LIN {X 5.728,Y -46.480,Z -106.471,A -90.000,B 90.000,C 0.000} C_DIS
LIN {X 5.220,Y -46.443,Z -106.628,A -90.000,B 90.000,C 0.000} C_DIS
LIN {X 4.791,Y -46.421,Z -106.762,A -90.000,B 90.000,C 0.000} C_DIS
LIN {X 4.548,Y -46.408,Z -106.845,A -90.000,B 90.000,C 0.000} C_DIS
LIN {X 4.247,Y -46.392,Z -106.952,A -90.000,B 90.000,C 0.000} C_DIS
LIN {X 3.683,Y -46.360,Z -107.175,A -90.000,B 90.000,C 0.000} C_DIS
LIN {X 3.330,Y -46.340,Z -107.324,A -90.000,B 90.000,C 0.000} C_DIS
LIN {X 2.924,Y -46.316,Z -107.512,A -90.000,B 90.000,C 0.000} C_DIS
LIN {X 2.654,Y -46.295,Z -107.645,A -90.000,B 90.000,C 0.000} C_DIS
LIN {X 1.447,Y -46.195,Z -108.262,A -90.000,B 90.000,C 0.000} C_DIS
LIN {X -0.684,Y -46.006,Z -109.354,A -90.000,B 90.000,C 0.000} C_DIS
LIN {X -0.987,Y -45.980,Z -109.516,A -90.000,B 90.000,C 0.000} C_DIS
LIN {X -1.310,Y -45.954,Z -109.697,A -90.000,B 90.000,C 0.000} C_DIS
LIN {X -1.716,Y -45.921,Z -109.939,A -90.000,B 90.000,C 0.000} C_DIS
LIN {X -2.229,Y -45.880,Z -110.266,A -90.000,B 90.000,C 0.000} C_DIS
LIN {X -2.497,Y -45.855,Z -110.452,A -90.000,B 90.000,C 0.000} C_DIS
LIN {X -4.271,Y -45.671,Z -111.693,A -90.000,B 90.000,C 0.000} C_DIS
LIN {X -4.661,Y -45.624,Z -111.967,A -90.000,B 90.000,C 0.000} C_DIS
LIN {X -5.221,Y -45.555,Z -112.383,A -90.000,B 90.000,C 0.000} C_DIS
LIN {X -5.480,Y -45.523,Z -112.584,A -90.000,B 90.000,C 0.000} C_DIS
LIN {X -5.669,Y -45.500,Z -112.740,A -90.000,B 90.000,C 0.000} C_DIS
LIN {X -5.871,Y -45.470,Z -112.907,A -90.000,B 90.000,C 0.000} C_DIS
LIN {X -6.143,Y -45.427,Z -113.144,A -90.000,B 90.000,C 0.000} C_DIS
LIN {X -6.336,Y -45.396,Z -113.323,A -90.000,B 90.000,C 0.000} C_DIS
LIN {X -7.007,Y -45.308,Z -113.952,A -90.000,B 90.000,C 0.000} C_DIS
LIN {X -7.165,Y -45.288,Z -114.092,A -90.000,B 90.000,C 0.000} C_DIS
LIN {X -7.242,Y -45.278,Z -114.154,A -90.000,B 90.000,C 0.000} C_DIS
LIN {X -7.389,Y -45.260,Z -114.260,A -90.000,B 90.000,C 0.000} C_DIS
LIN {X -7.460,Y -45.251,Z -114.305,A -90.000,B 90.000,C 0.000} C_DIS
LIN {X -7.595,Y -45.234,Z -114.380,A -90.000,B 90.000,C 0.000} C_DIS
LIN {X -7.660,Y -45.226,Z -114.410,A -90.000,B 90.000,C 0.000} C_DIS
LIN {X -7.783,Y -45.212,Z -114.455,A -90.000,B 90.000,C 0.000} C_DIS
LIN {X -7.869,Y -45.202,Z -114.476,A -90.000,B 90.000,C 0.000} C_DIS
LIN {X -7.951,Y -45.193,Z -114.487,A -90.000,B 90.000,C 0.000} C_DIS
LIN {X -8.029,Y -45.184,Z -114.489,A -90.000,B 90.000,C 0.000} C_DIS
LIN {X -8.077,Y -45.179,Z -114.485,A -90.000,B 90.000,C 0.000} C_DIS
LIN {X -8.124,Y -45.174,Z -114.476,A -90.000,B 90.000,C 0.000} C_DIS
LIN {X -8.189,Y -45.167,Z -114.456,A -90.000,B 90.000,C 0.000} C_DIS
LIN {X -8.249,Y -45.161,Z -114.428,A -90.000,B 90.000,C 0.000} C_DIS
LIN {X -8.305,Y -45.156,Z -114.391,A -90.000,B 90.000,C 0.000} C_DIS
LIN {X -8.338,Y -45.153,Z -114.363,A -90.000,B 90.000,C 0.000} C_DIS
LIN {X -8.370,Y -45.150,Z -114.331,A -90.000,B 90.000,C 0.000} C_DIS
LIN {X -8.425,Y -45.146,Z -114.257,A -90.000,B 90.000,C 0.000} C_DIS
LIN {X -8.450,Y -45.144,Z -114.216,A -90.000,B 90.000,C 0.000} C_DIS
LIN {X -8.490,Y -45.142,Z -114.125,A -90.000,B 90.000,C 0.000} C_DIS
LIN {X -8.507,Y -45.141,Z -114.075,A -90.000,B 90.000,C 0.000} C_DIS
LIN {X -8.533,Y -45.140,Z -113.968,A -90.000,B 90.000,C 0.000} C_DIS
LIN {X -8.548,Y -45.141,Z -113.852,A -90.000,B 90.000,C 0.000} C_DIS
LIN {X -8.552,Y -45.142,Z -113.791,A -90.000,B 90.000,C 0.000} C_DIS
LIN {X -8.552,Y -45.145,Z -113.662,A -90.000,B 90.000,C 0.000} C_DIS
LIN {X -8.547,Y -45.147,Z -113.595,A -90.000,B 90.000,C 0.000} C_DIS
LIN {X -8.531,Y -45.151,Z -113.457,A -90.000,B 90.000,C 0.000} C_DIS
LIN {X -8.518,Y -45.154,Z -113.385,A -90.000,B 90.000,C 0.000} C_DIS
LIN {X -8.485,Y -45.161,Z -113.238,A -90.000,B 90.000,C 0.000} C_DIS
LIN {X -8.464,Y -45.165,Z -113.163,A -90.000,B 90.000,C 0.000} C_DIS
LIN {X -8.414,Y -45.173,Z -113.010,A -90.000,B 90.000,C 0.000} C_DIS
LIN {X -8.352,Y -45.183,Z -112.854,A -90.000,B 90.000,C 0.000} C_DIS
LIN {X -8.316,Y -45.188,Z -112.775,A -90.000,B 90.000,C 0.000} C_DIS
LIN {X -8.236,Y -45.200,Z -112.616,A -90.000,B 90.000,C 0.000} C_DIS
LIN {X -8.145,Y -45.213,Z -112.456,A -90.000,B 90.000,C 0.000} C_DIS
LIN {X -8.040,Y -45.228,Z -112.297,A -90.000,B 90.000,C 0.000} C_DIS
LIN {X -7.924,Y -45.243,Z -112.138,A -90.000,B 90.000,C 0.000} C_DIS
LIN {X -7.861,Y -45.252,Z -112.060,A -90.000,B 90.000,C 0.000} C_DIS
LIN {X -7.725,Y -45.271,Z -111.904,A -90.000,B 90.000,C 0.000} C_DIS
LIN {X -7.577,Y -45.290,Z -111.752,A -90.000,B 90.000,C 0.000} C_DIS
LIN {X -7.415,Y -45.308,Z -111.604,A -90.000,B 90.000,C 0.000} C_DIS
LIN {X -7.133,Y -45.343,Z -111.360,A -90.000,B 90.000,C 0.000} C_DIS
LIN {X -6.892,Y -45.373,Z -111.162,A -90.000,B 90.000,C 0.000} C_DIS
LIN {X -6.663,Y -45.406,Z -110.976,A -90.000,B 90.000,C 0.000} C_DIS
LIN {X -6.402,Y -45.443,Z -110.773,A -90.000,B 90.000,C 0.000} C_DIS
LIN {X -5.802,Y -45.528,Z -110.327,A -90.000,B 90.000,C 0.000} C_DIS
LIN {X -4.905,Y -45.651,Z -109.697,A -90.000,B 90.000,C 0.000} C_DIS
LIN {X -3.365,Y -45.832,Z -108.621,A -90.000,B 90.000,C 0.000} C_DIS
LIN {X -2.790,Y -45.899,Z -108.252,A -90.000,B 90.000,C 0.000} C_DIS
LIN {X -2.292,Y -45.956,Z -107.955,A -90.000,B 90.000,C 0.000} C_DIS
LIN {X -1.892,Y -46.001,Z -107.732,A -90.000,B 90.000,C 0.000} C_DIS
LIN {X -1.584,Y -46.032,Z -107.568,A -90.000,B 90.000,C 0.000} C_DIS
LIN {X 1.658,Y -46.324,Z -105.909,A -90.000,B 90.000,C 0.000} C_DIS
LIN {X 2.084,Y -46.370,Z -105.698,A -90.000,B 90.000,C 0.000} C_DIS
LIN {X 2.546,Y -46.419,Z -105.486,A -90.000,B 90.000,C 0.000} C_DIS
LIN {X 2.945,Y -46.458,Z -105.318,A -90.000,B 90.000,C 0.000} C_DIS
LIN {X 3.509,Y -46.508,Z -105.097,A -90.000,B 90.000,C 0.000} C_DIS
LIN {X 3.902,Y -46.541,Z -104.957,A -90.000,B 90.000,C 0.000} C_DIS
LIN {X 4.190,Y -46.565,Z -104.860,A -90.000,B 90.000,C 0.000} C_DIS
LIN {X 4.953,Y -46.625,Z -104.624,A -90.000,B 90.000,C 0.000} C_DIS
LIN {X 5.350,Y -46.652,Z -104.500,A -90.000,B 90.000,C 0.000} C_DIS
LIN {X 7.425,Y -46.782,Z -103.856,A -90.000,B 90.000,C 0.000} C_DIS
LIN {X 9.167,Y -46.887,Z -103.318,A -90.000,B 90.000,C 0.000} C_DIS
LIN {X 9.792,Y -46.919,Z -103.138,A -90.000,B 90.000,C 0.000} C_DIS
LIN {X 10.236,Y -46.939,Z -103.026,A -90.000,B 90.000,C 0.000} C_DIS
LIN {X 10.412,Y -46.943,Z -102.982,A -90.000,B 90.000,C 0.000} C_DIS
LIN {X 10.698,Y -46.949,Z -102.919,A -90.000,B 90.000,C 0.000} C_DIS
LIN {X 11.087,Y -46.957,Z -102.840,A -90.000,B 90.000,C 0.000} C_DIS
LIN {X 11.780,Y -46.971,Z -102.720,A -90.000,B 90.000,C 0.000} C_DIS
LIN {X 12.175,Y -46.978,Z -102.667,A -90.000,B 90.000,C 0.000} C_DIS
LIN {X 14.089,Y -47.019,Z -102.461,A -90.000,B 90.000,C 0.000} C_DIS
LIN {X 16.194,Y -47.092,Z -102.235,A -90.000,B 90.000,C 0.000} C_DIS
LIN {X 16.820,Y -47.105,Z -102.168,A -90.000,B 90.000,C 0.000} C_DIS
LIN {X 17.411,Y -47.109,Z -102.121,A -90.000,B 90.000,C 0.000} C_DIS
LIN {X 17.868,Y -47.112,Z -102.099,A -90.000,B 90.000,C 0.000} C_DIS
LIN {X 18.326,Y -47.118,Z -102.089,A -90.000,B 90.000,C 0.000} C_DIS
LIN {X 19.084,Y -47.128,Z -102.091,A -90.000,B 90.000,C 0.000} C_DIS
LIN {X 19.404,Y -47.133,Z -102.102,A -90.000,B 90.000,C 0.000} C_DIS
LIN {X 19.767,Y -47.139,Z -102.122,A -90.000,B 90.000,C 0.000} C_DIS
LIN {X 20.317,Y -47.149,Z -102.167,A -90.000,B 90.000,C 0.000} C_DIS
LIN {X 20.522,Y -47.153,Z -102.188,A -90.000,B 90.000,C 0.000} C_DIS
LIN {X 20.920,Y -47.161,Z -102.234,A -90.000,B 90.000,C 0.000} C_DIS
LIN {X 21.317,Y -47.169,Z -102.291,A -90.000,B 90.000,C 0.000} C_DIS
LIN {X 21.583,Y -47.172,Z -102.331,A -90.000,B 90.000,C 0.000} C_DIS
LIN {X 23.495,Y -47.194,Z -102.667,A -90.000,B 90.000,C 0.000} C_DIS
LIN {X 24.740,Y -47.209,Z -102.887,A -90.000,B 90.000,C 0.000} C_DIS
LIN {X 24.965,Y -47.205,Z -102.927,A -90.000,B 90.000,C 0.000} C_DIS
LIN {X 25.904,Y -47.190,Z -103.117,A -90.000,B 90.000,C 0.000} C_DIS
LIN {X 26.315,Y -47.185,Z -103.209,A -90.000,B 90.000,C 0.000} C_DIS
LIN {X 26.791,Y -47.182,Z -103.331,A -90.000,B 90.000,C 0.000} C_DIS
LIN {X 27.008,Y -47.182,Z -103.392,A -90.000,B 90.000,C 0.000} C_DIS
LIN {X 27.382,Y -47.180,Z -103.502,A -90.000,B 90.000,C 0.000} C_DIS
LIN {X 27.937,Y -47.180,Z -103.682,A -90.000,B 90.000,C 0.000} C_DIS
LIN {X 28.105,Y -47.179,Z -103.743,A -90.000,B 90.000,C 0.000} C_DIS
LIN {X 28.411,Y -47.164,Z -103.857,A -90.000,B 90.000,C 0.000} C_DIS
LIN {X 28.662,Y -47.153,Z -103.956,A -90.000,B 90.000,C 0.000} C_DIS
LIN {X 28.872,Y -47.143,Z -104.045,A -90.000,B 90.000,C 0.000} C_DIS
LIN {X 29.063,Y -47.134,Z -104.130,A -90.000,B 90.000,C 0.000} C_DIS
LIN {X 29.386,Y -47.126,Z -104.275,A -90.000,B 90.000,C 0.000} C_DIS
LIN {X 29.815,Y -47.115,Z -104.478,A -90.000,B 90.000,C 0.000} C_DIS
LIN {X 30.271,Y -47.106,Z -104.714,A -90.000,B 90.000,C 0.000} C_DIS
LIN {X 30.581,Y -47.100,Z -104.885,A -90.000,B 90.000,C 0.000} C_DIS
LIN {X 30.945,Y -47.093,Z -105.100,A -90.000,B 90.000,C 0.000} C_DIS
LIN {X 31.194,Y -47.089,Z -105.254,A -90.000,B 90.000,C 0.000} C_DIS
LIN {X 31.416,Y -47.085,Z -105.399,A -90.000,B 90.000,C 0.000} C_DIS
LIN {X 31.625,Y -47.072,Z -105.535,A -90.000,B 90.000,C 0.000} C_DIS
LIN {X 31.892,Y -47.053,Z -105.721,A -90.000,B 90.000,C 0.000} C_DIS
LIN {X 32.034,Y -47.043,Z -105.821,A -90.000,B 90.000,C 0.000} C_DIS
LIN {X 32.303,Y -47.018,Z -106.021,A -90.000,B 90.000,C 0.000} C_DIS
LIN {X 33.453,Y -46.911,Z -106.918,A -90.000,B 90.000,C 0.000} C_DIS
LIN {X 34.289,Y -46.869,Z -107.570,A -90.000,B 90.000,C 0.000} C_DIS
LIN {X 34.659,Y -46.837,Z -107.865,A -90.000,B 90.000,C 0.000} C_DIS
LIN {X 35.145,Y -46.771,Z -108.283,A -90.000,B 90.000,C 0.000} C_DIS
LIN {X 35.492,Y -46.725,Z -108.600,A -90.000,B 90.000,C 0.000} C_DIS
LIN {X 35.573,Y -46.718,Z -108.676,A -90.000,B 90.000,C 0.000} C_DIS
LIN {X 35.836,Y -46.694,Z -108.932,A -90.000,B 90.000,C 0.000} C_DIS
LIN {X 36.071,Y -46.673,Z -109.170,A -90.000,B 90.000,C 0.000} C_DIS
LIN {X 36.256,Y -46.656,Z -109.365,A -90.000,B 90.000,C 0.000} C_DIS
LIN {X 36.535,Y -46.631,Z -109.672,A -90.000,B 90.000,C 0.000} C_DIS
LIN {X 36.869,Y -46.601,Z -110.055,A -90.000,B 90.000,C 0.000} C_DIS
LIN {X 37.225,Y -46.559,Z -110.463,A -90.000,B 90.000,C 0.000} C_DIS
LIN {X 37.348,Y -46.546,Z -110.604,A -90.000,B 90.000,C 0.000} C_DIS
LIN {X 37.484,Y -46.518,Z -110.763,A -90.000,B 90.000,C 0.000} C_DIS
LIN {X 37.843,Y -46.443,Z -111.213,A -90.000,B 90.000,C 0.000} C_DIS
LIN {X 38.185,Y -46.371,Z -111.667,A -90.000,B 90.000,C 0.000} C_DIS
LIN {X 38.452,Y -46.313,Z -112.050,A -90.000,B 90.000,C 0.000} C_DIS
LIN {X 38.592,Y -46.282,Z -112.262,A -90.000,B 90.000,C 0.000} C_DIS
LIN {X 38.702,Y -46.264,Z -112.429,A -90.000,B 90.000,C 0.000} C_DIS
LIN {X 39.009,Y -46.212,Z -112.929,A -90.000,B 90.000,C 0.000} C_DIS
LIN {X 39.264,Y -46.169,Z -113.380,A -90.000,B 90.000,C 0.000} C_DIS
LIN {X 39.457,Y -46.135,Z -113.750,A -90.000,B 90.000,C 0.000} C_DIS
LIN {X 39.482,Y -46.131,Z -113.800,A -90.000,B 90.000,C 0.000} C_DIS
LIN {X 39.697,Y -46.073,Z -114.238,A -90.000,B 90.000,C 0.000} C_DIS
LIN {X 39.731,Y -46.063,Z -114.313,A -90.000,B 90.000,C 0.000} C_DIS
LIN {X 39.924,Y -45.993,Z -114.757,A -90.000,B 90.000,C 0.000} C_DIS
LIN {X 40.070,Y -45.936,Z -115.126,A -90.000,B 90.000,C 0.000} C_DIS
LIN {X 40.157,Y -45.898,Z -115.357,A -90.000,B 90.000,C 0.000} C_DIS
LIN {X 40.283,Y -45.841,Z -115.720,A -90.000,B 90.000,C 0.000} C_DIS
LIN {X 40.401,Y -45.785,Z -116.075,A -90.000,B 90.000,C 0.000} C_DIS
LIN {X 40.525,Y -45.724,Z -116.487,A -90.000,B 90.000,C 0.000} C_DIS
LIN {X 40.608,Y -45.681,Z -116.782,A -90.000,B 90.000,C 0.000} C_DIS
LIN {X 40.716,Y -45.622,Z -117.213,A -90.000,B 90.000,C 0.000} C_DIS
LIN {X 40.827,Y -45.556,Z -117.712,A -90.000,B 90.000,C 0.000} C_DIS
LIN {X 40.882,Y -45.522,Z -117.974,A -90.000,B 90.000,C 0.000} C_DIS
LIN {X 40.917,Y -45.497,Z -118.175,A -90.000,B 90.000,C 0.000} C_DIS
LIN {X 41.005,Y -45.406,Z -118.721,A -90.000,B 90.000,C 0.000} C_DIS
LIN {X 41.031,Y -45.377,Z -118.893,A -90.000,B 90.000,C 0.000} C_DIS
LIN {X 41.089,Y -45.308,Z -119.275,A -90.000,B 90.000,C 0.000} C_DIS
LIN {X 41.089,Y -60.000,Z -119.275,A -90.000,B 90.000,C 0.000} C_DIS
LIN {X -8.114,Y -60.000,Z -109.579,A -90.000,B 90.000,C 0.000} C_DIS
LIN {X -8.114,Y -45.308,Z -109.579,A -90.000,B 90.000,C 0.000} C_DIS
LIN {X -7.884,Y -45.344,Z -109.393,A -90.000,B 90.000,C 0.000} C_DIS
LIN {X -7.589,Y -45.390,Z -109.164,A -90.000,B 90.000,C 0.000} C_DIS
LIN {X -6.942,Y -45.489,Z -108.685,A -90.000,B 90.000,C 0.000} C_DIS
LIN {X -5.499,Y -45.679,Z -107.673,A -90.000,B 90.000,C 0.000} C_DIS
LIN {X -4.509,Y -45.809,Z -106.981,A -90.000,B 90.000,C 0.000} C_DIS
LIN {X -4.274,Y -45.840,Z -106.828,A -90.000,B 90.000,C 0.000} C_DIS
LIN {X -3.813,Y -45.895,Z -106.533,A -90.000,B 90.000,C 0.000} C_DIS
LIN {X -3.268,Y -45.958,Z -106.209,A -90.000,B 90.000,C 0.000} C_DIS
LIN {X -2.830,Y -46.009,Z -105.965,A -90.000,B 90.000,C 0.000} C_DIS
LIN {X -2.497,Y -46.046,Z -105.789,A -90.000,B 90.000,C 0.000} C_DIS
LIN {X -1.090,Y -46.212,Z -105.069,A -90.000,B 90.000,C 0.000} C_DIS
LIN {X 0.519,Y -46.415,Z -104.248,A -90.000,B 90.000,C 0.000} C_DIS
LIN {X 0.761,Y -46.443,Z -104.125,A -90.000,B 90.000,C 0.000} C_DIS
LIN {X 1.242,Y -46.495,Z -103.888,A -90.000,B 90.000,C 0.000} C_DIS
LIN {X 1.630,Y -46.534,Z -103.710,A -90.000,B 90.000,C 0.000} C_DIS
LIN {X 1.762,Y -46.547,Z -103.651,A -90.000,B 90.000,C 0.000} C_DIS
LIN {X 2.207,Y -46.585,Z -103.464,A -90.000,B 90.000,C 0.000} C_DIS
LIN {X 2.834,Y -46.637,Z -103.219,A -90.000,B 90.000,C 0.000} C_DIS
LIN {X 3.259,Y -46.670,Z -103.067,A -90.000,B 90.000,C 0.000} C_DIS
LIN {X 3.630,Y -46.699,Z -102.945,A -90.000,B 90.000,C 0.000} C_DIS
LIN {X 5.478,Y -46.844,Z -102.372,A -90.000,B 90.000,C 0.000} C_DIS
LIN {X 6.367,Y -46.906,Z -102.097,A -90.000,B 90.000,C 0.000} C_DIS
LIN {X 8.611,Y -46.960,Z -101.398,A -90.000,B 90.000,C 0.000} C_DIS
LIN {X 9.301,Y -46.982,Z -101.200,A -90.000,B 90.000,C 0.000} C_DIS
LIN {X 9.980,Y -47.002,Z -101.031,A -90.000,B 90.000,C 0.000} C_DIS
LIN {X 10.298,Y -47.011,Z -100.961,A -90.000,B 90.000,C 0.000} C_DIS
LIN {X 10.746,Y -47.017,Z -100.870,A -90.000,B 90.000,C 0.000} C_DIS
LIN {X 10.940,Y -47.018,Z -100.837,A -90.000,B 90.000,C 0.000} C_DIS
LIN {X 11.512,Y -47.006,Z -100.739,A -90.000,B 90.000,C 0.000} C_DIS
LIN {X 11.961,Y -46.997,Z -100.679,A -90.000,B 90.000,C 0.000} C_DIS
LIN {X 13.433,Y -46.972,Z -100.521,A -90.000,B 90.000,C 0.000} C_DIS
LIN {X 14.968,Y -46.961,Z -100.358,A -90.000,B 90.000,C 0.000} C_DIS
LIN {X 16.661,Y -46.970,Z -100.179,A -90.000,B 90.000,C 0.000} C_DIS
LIN {X 17.319,Y -46.974,Z -100.127,A -90.000,B 90.000,C 0.000} C_DIS
LIN {X 17.825,Y -46.979,Z -100.104,A -90.000,B 90.000,C 0.000} C_DIS
LIN {X 18.333,Y -46.983,Z -100.094,A -90.000,B 90.000,C 0.000} C_DIS
LIN {X 19.153,Y -46.992,Z -100.097,A -90.000,B 90.000,C 0.000} C_DIS
LIN {X 19.518,Y -46.997,Z -100.110,A -90.000,B 90.000,C 0.000} C_DIS
LIN {X 19.880,Y -47.000,Z -100.130,A -90.000,B 90.000,C 0.000} C_DIS
LIN {X 20.522,Y -47.003,Z -100.183,A -90.000,B 90.000,C 0.000} C_DIS
LIN {X 20.751,Y -47.005,Z -100.207,A -90.000,B 90.000,C 0.000} C_DIS
LIN {X 21.210,Y -47.009,Z -100.261,A -90.000,B 90.000,C 0.000} C_DIS
LIN {X 21.930,Y -47.021,Z -100.367,A -90.000,B 90.000,C 0.000} C_DIS
LIN {X 25.371,Y -47.046,Z -100.975,A -90.000,B 90.000,C 0.000} C_DIS
LIN {X 26.337,Y -47.032,Z -101.171,A -90.000,B 90.000,C 0.000} C_DIS
LIN {X 26.812,Y -47.026,Z -101.278,A -90.000,B 90.000,C 0.000} C_DIS
LIN {X 27.327,Y -47.024,Z -101.411,A -90.000,B 90.000,C 0.000} C_DIS
LIN {X 27.568,Y -47.024,Z -101.479,A -90.000,B 90.000,C 0.000} C_DIS
LIN {X 27.999,Y -47.024,Z -101.606,A -90.000,B 90.000,C 0.000} C_DIS
LIN {X 28.616,Y -47.028,Z -101.807,A -90.000,B 90.000,C 0.000} C_DIS
LIN {X 28.870,Y -47.031,Z -101.899,A -90.000,B 90.000,C 0.000} C_DIS
LIN {X 29.159,Y -47.023,Z -102.007,A -90.000,B 90.000,C 0.000} C_DIS
LIN {X 29.594,Y -47.011,Z -102.184,A -90.000,B 90.000,C 0.000} C_DIS
LIN {X 30.164,Y -46.987,Z -102.437,A -90.000,B 90.000,C 0.000} C_DIS
LIN {X 30.649,Y -46.967,Z -102.665,A -90.000,B 90.000,C 0.000} C_DIS
LIN {X 30.730,Y -46.964,Z -102.705,A -90.000,B 90.000,C 0.000} C_DIS
LIN {X 31.158,Y -46.948,Z -102.928,A -90.000,B 90.000,C 0.000} C_DIS
LIN {X 31.528,Y -46.933,Z -103.131,A -90.000,B 90.000,C 0.000} C_DIS
LIN {X 31.702,Y -46.926,Z -103.233,A -90.000,B 90.000,C 0.000} C_DIS
LIN {X 32.007,Y -46.921,Z -103.414,A -90.000,B 90.000,C 0.000} C_DIS
LIN {X 32.240,Y -46.917,Z -103.558,A -90.000,B 90.000,C 0.000} C_DIS
LIN {X 32.365,Y -46.911,Z -103.639,A -90.000,B 90.000,C 0.000} C_DIS
LIN {X 32.699,Y -46.886,Z -103.859,A -90.000,B 90.000,C 0.000} C_DIS
LIN {X 33.038,Y -46.861,Z -104.092,A -90.000,B 90.000,C 0.000} C_DIS
LIN {X 33.212,Y -46.848,Z -104.217,A -90.000,B 90.000,C 0.000} C_DIS
LIN {X 33.517,Y -46.827,Z -104.443,A -90.000,B 90.000,C 0.000} C_DIS
LIN {X 33.622,Y -46.819,Z -104.524,A -90.000,B 90.000,C 0.000} C_DIS
LIN {X 35.278,Y -46.750,Z -105.810,A -90.000,B 90.000,C 0.000} C_DIS
LIN {X 35.408,Y -46.740,Z -105.912,A -90.000,B 90.000,C 0.000} C_DIS
LIN {X 35.682,Y -46.709,Z -106.130,A -90.000,B 90.000,C 0.000} C_DIS
LIN {X 35.947,Y -46.685,Z -106.343,A -90.000,B 90.000,C 0.000} C_DIS
LIN {X 36.318,Y -46.653,Z -106.660,A -90.000,B 90.000,C 0.000} C_DIS
LIN {X 36.503,Y -46.632,Z -106.821,A -90.000,B 90.000,C 0.000} C_DIS
LIN {X 36.799,Y -46.594,Z -107.092,A -90.000,B 90.000,C 0.000} C_DIS
LIN {X 36.957,Y -46.573,Z -107.240,A -90.000,B 90.000,C 0.000} C_DIS
LIN {X 37.247,Y -46.533,Z -107.523,A -90.000,B 90.000,C 0.000} C_DIS
LIN {X 37.504,Y -46.498,Z -107.786,A -90.000,B 90.000,C 0.000} C_DIS
LIN {X 37.594,Y -46.485,Z -107.881,A -90.000,B 90.000,C 0.000} C_DIS
LIN {X 37.795,Y -46.467,Z -108.097,A -90.000,B 90.000,C 0.000} C_DIS
LIN {X 38.003,Y -46.449,Z -108.327,A -90.000,B 90.000,C 0.000} C_DIS
LIN {X 38.230,Y -46.427,Z -108.586,A -90.000,B 90.000,C 0.000} C_DIS
LIN {X 38.994,Y -46.276,Z -109.475,A -90.000,B 90.000,C 0.000} C_DIS
LIN {X 39.114,Y -46.252,Z -109.623,A -90.000,B 90.000,C 0.000} C_DIS
LIN {X 39.376,Y -46.210,Z -109.949,A -90.000,B 90.000,C 0.000} C_DIS
LIN {X 39.757,Y -46.150,Z -110.450,A -90.000,B 90.000,C 0.000} C_DIS
LIN {X 40.091,Y -46.098,Z -110.924,A -90.000,B 90.000,C 0.000} C_DIS
LIN {X 40.341,Y -46.059,Z -111.302,A -90.000,B 90.000,C 0.000} C_DIS
LIN {X 40.423,Y -46.046,Z -111.431,A -90.000,B 90.000,C 0.000} C_DIS
LIN {X 40.592,Y -46.013,Z -111.707,A -90.000,B 90.000,C 0.000} C_DIS
LIN {X 40.728,Y -45.979,Z -111.934,A -90.000,B 90.000,C 0.000} C_DIS
LIN {X 40.865,Y -45.942,Z -112.180,A -90.000,B 90.000,C 0.000} C_DIS
LIN {X 41.010,Y -45.893,Z -112.444,A -90.000,B 90.000,C 0.000} C_DIS
LIN {X 41.238,Y -45.814,Z -112.897,A -90.000,B 90.000,C 0.000} C_DIS
LIN {X 41.475,Y -45.731,Z -113.388,A -90.000,B 90.000,C 0.000} C_DIS
LIN {X 41.735,Y -45.636,Z -113.988,A -90.000,B 90.000,C 0.000} C_DIS
LIN {X 41.933,Y -45.560,Z -114.493,A -90.000,B 90.000,C 0.000} C_DIS
LIN {X 41.996,Y -45.535,Z -114.659,A -90.000,B 90.000,C 0.000} C_DIS
LIN {X 42.157,Y -45.470,Z -115.121,A -90.000,B 90.000,C 0.000} C_DIS
LIN {X 42.269,Y -45.424,Z -115.458,A -90.000,B 90.000,C 0.000} C_DIS
LIN {X 42.371,Y -45.380,Z -115.792,A -90.000,B 90.000,C 0.000} C_DIS
LIN {X 42.432,Y -45.346,Z -116.004,A -90.000,B 90.000,C 0.000} C_DIS
LIN {X 42.496,Y -45.308,Z -116.235,A -90.000,B 90.000,C 0.000} C_DIS
LIN {X 42.496,Y -60.000,Z -116.235,A -90.000,B 90.000,C 0.000} C_DIS
LIN {X -8.899,Y -60.000,Z -107.650,A -90.000,B 90.000,C 0.000} C_DIS
LIN {X -8.899,Y -45.308,Z -107.650,A -90.000,B 90.000,C 0.000} C_DIS
LIN {X -8.772,Y -45.328,Z -107.553,A -90.000,B 90.000,C 0.000} C_DIS
LIN {X -8.085,Y -45.431,Z -107.044,A -90.000,B 90.000,C 0.000} C_DIS
LIN {X -7.649,Y -45.496,Z -106.738,A -90.000,B 90.000,C 0.000} C_DIS
LIN {X -6.645,Y -45.653,Z -106.034,A -90.000,B 90.000,C 0.000} C_DIS
LIN {X -5.599,Y -45.811,Z -105.304,A -90.000,B 90.000,C 0.000} C_DIS
LIN {X -5.136,Y -45.879,Z -105.005,A -90.000,B 90.000,C 0.000} C_DIS
LIN {X -4.837,Y -45.923,Z -104.815,A -90.000,B 90.000,C 0.000} C_DIS
LIN {X -4.234,Y -46.000,Z -104.459,A -90.000,B 90.000,C 0.000} C_DIS
LIN {X -3.770,Y -46.057,Z -104.200,A -90.000,B 90.000,C 0.000} C_DIS
LIN {X -3.412,Y -46.103,Z -104.011,A -90.000,B 90.000,C 0.000} C_DIS
LIN {X -0.893,Y -46.422,Z -102.725,A -90.000,B 90.000,C 0.000} C_DIS
LIN {X -0.128,Y -46.501,Z -102.334,A -90.000,B 90.000,C 0.000} C_DIS
LIN {X 0.060,Y -46.520,Z -102.242,A -90.000,B 90.000,C 0.000} C_DIS
LIN {X 0.404,Y -46.559,Z -102.073,A -90.000,B 90.000,C 0.000} C_DIS
LIN {X 0.936,Y -46.618,Z -101.831,A -90.000,B 90.000,C 0.000} C_DIS
LIN {X 1.473,Y -46.677,Z -101.606,A -90.000,B 90.000,C 0.000} C_DIS
LIN {X 2.155,Y -46.749,Z -101.341,A -90.000,B 90.000,C 0.000} C_DIS
LIN {X 2.551,Y -46.782,Z -101.200,A -90.000,B 90.000,C 0.000} C_DIS
LIN {X 2.691,Y -46.792,Z -101.152,A -90.000,B 90.000,C 0.000} C_DIS
LIN {X 3.031,Y -46.805,Z -101.039,A -90.000,B 90.000,C 0.000} C_DIS
LIN {X 4.884,Y -46.867,Z -100.463,A -90.000,B 90.000,C 0.000} C_DIS
LIN {X 5.389,Y -46.890,Z -100.306,A -90.000,B 90.000,C 0.000} C_DIS
LIN {X 6.585,Y -46.942,Z -99.934,A -90.000,B 90.000,C 0.000} C_DIS
LIN {X 6.830,Y -46.946,Z -99.858,A -90.000,B 90.000,C 0.000} C_DIS
LIN {X 7.436,Y -46.940,Z -99.669,A -90.000,B 90.000,C 0.000} C_DIS
LIN {X 8.062,Y -46.918,Z -99.475,A -90.000,B 90.000,C 0.000} C_DIS
LIN {X 8.820,Y -46.892,Z -99.261,A -90.000,B 90.000,C 0.000} C_DIS
LIN {X 9.554,Y -46.869,Z -99.081,A -90.000,B 90.000,C 0.000} C_DIS
LIN {X 9.905,Y -46.862,Z -99.005,A -90.000,B 90.000,C 0.000} C_DIS
LIN {X 10.407,Y -46.855,Z -98.906,A -90.000,B 90.000,C 0.000} C_DIS
LIN {X 11.244,Y -46.845,Z -98.763,A -90.000,B 90.000,C 0.000} C_DIS
LIN {X 11.745,Y -46.840,Z -98.697,A -90.000,B 90.000,C 0.000} C_DIS
LIN {X 12.793,Y -46.828,Z -98.584,A -90.000,B 90.000,C 0.000} C_DIS
LIN {X 14.289,Y -46.761,Z -98.429,A -90.000,B 90.000,C 0.000} C_DIS
LIN {X 15.106,Y -46.718,Z -98.347,A -90.000,B 90.000,C 0.000} C_DIS
LIN {X 15.976,Y -46.685,Z -98.261,A -90.000,B 90.000,C 0.000} C_DIS
LIN {X 16.507,Y -46.666,Z -98.208,A -90.000,B 90.000,C 0.000} C_DIS
LIN {X 17.232,Y -46.645,Z -98.157,A -90.000,B 90.000,C 0.000} C_DIS
LIN {X 17.788,Y -46.633,Z -98.135,A -90.000,B 90.000,C 0.000} C_DIS
LIN {X 18.344,Y -46.627,Z -98.126,A -90.000,B 90.000,C 0.000} C_DIS
LIN {X 19.227,Y -46.620,Z -98.133,A -90.000,B 90.000,C 0.000} C_DIS
LIN {X 19.632,Y -46.617,Z -98.149,A -90.000,B 90.000,C 0.000} C_DIS
LIN {X 20.045,Y -46.617,Z -98.174,A -90.000,B 90.000,C 0.000} C_DIS
LIN {X 20.727,Y -46.620,Z -98.231,A -90.000,B 90.000,C 0.000} C_DIS
LIN {X 21.018,Y -46.623,Z -98.262,A -90.000,B 90.000,C 0.000} C_DIS
LIN {X 21.504,Y -46.629,Z -98.319,A -90.000,B 90.000,C 0.000} C_DIS
LIN {X 21.929,Y -46.637,Z -98.382,A -90.000,B 90.000,C 0.000} C_DIS
LIN {X 22.273,Y -46.644,Z -98.434,A -90.000,B 90.000,C 0.000} C_DIS
LIN {X 22.575,Y -46.649,Z -98.486,A -90.000,B 90.000,C 0.000} C_DIS
LIN {X 25.715,Y -46.674,Z -99.040,A -90.000,B 90.000,C 0.000} C_DIS
LIN {X 26.009,Y -46.678,Z -99.098,A -90.000,B 90.000,C 0.000} C_DIS
LIN {X 26.766,Y -46.666,Z -99.252,A -90.000,B 90.000,C 0.000} C_DIS
LIN {X 27.303,Y -46.661,Z -99.374,A -90.000,B 90.000,C 0.000} C_DIS
LIN {X 27.857,Y -46.658,Z -99.518,A -90.000,B 90.000,C 0.000} C_DIS
LIN {X 28.123,Y -46.657,Z -99.593,A -90.000,B 90.000,C 0.000} C_DIS
LIN {X 28.612,Y -46.658,Z -99.737,A -90.000,B 90.000,C 0.000} C_DIS
LIN {X 29.292,Y -46.663,Z -99.961,A -90.000,B 90.000,C 0.000} C_DIS
LIN {X 29.544,Y -46.665,Z -100.052,A -90.000,B 90.000,C 0.000} C_DIS
LIN {X 29.920,Y -46.655,Z -100.194,A -90.000,B 90.000,C 0.000} C_DIS
LIN {X 30.381,Y -46.646,Z -100.382,A -90.000,B 90.000,C 0.000} C_DIS
LIN {X 31.015,Y -46.636,Z -100.662,A -90.000,B 90.000,C 0.000} C_DIS
LIN {X 31.570,Y -46.630,Z -100.921,A -90.000,B 90.000,C 0.000} C_DIS
LIN {X 32.100,Y -46.629,Z -101.193,A -90.000,B 90.000,C 0.000} C_DIS
LIN {X 32.542,Y -46.631,Z -101.434,A -90.000,B 90.000,C 0.000} C_DIS
LIN {X 32.878,Y -46.634,Z -101.630,A -90.000,B 90.000,C 0.000} C_DIS
LIN {X 33.078,Y -46.631,Z -101.749,A -90.000,B 90.000,C 0.000} C_DIS
LIN {X 33.370,Y -46.622,Z -101.933,A -90.000,B 90.000,C 0.000} C_DIS
LIN {X 33.811,Y -46.610,Z -102.219,A -90.000,B 90.000,C 0.000} C_DIS
LIN {X 34.152,Y -46.603,Z -102.452,A -90.000,B 90.000,C 0.000} C_DIS
LIN {X 34.467,Y -46.598,Z -102.676,A -90.000,B 90.000,C 0.000} C_DIS
LIN {X 34.726,Y -46.593,Z -102.867,A -90.000,B 90.000,C 0.000} C_DIS
LIN {X 35.254,Y -46.585,Z -103.275,A -90.000,B 90.000,C 0.000} C_DIS
LIN {X 35.458,Y -46.575,Z -103.434,A -90.000,B 90.000,C 0.000} C_DIS
LIN {X 35.809,Y -46.551,Z -103.707,A -90.000,B 90.000,C 0.000} C_DIS
LIN {X 36.093,Y -46.538,Z -103.928,A -90.000,B 90.000,C 0.000} C_DIS
LIN {X 36.197,Y -46.529,Z -104.009,A -90.000,B 90.000,C 0.000} C_DIS
LIN {X 36.910,Y -46.447,Z -104.573,A -90.000,B 90.000,C 0.000} C_DIS
LIN {X 37.221,Y -46.412,Z -104.825,A -90.000,B 90.000,C 0.000} C_DIS
LIN {X 37.761,Y -46.353,Z -105.291,A -90.000,B 90.000,C 0.000} C_DIS
LIN {X 38.172,Y -46.319,Z -105.664,A -90.000,B 90.000,C 0.000} C_DIS
LIN {X 38.326,Y -46.306,Z -105.806,A -90.000,B 90.000,C 0.000} C_DIS
LIN {X 38.646,Y -46.281,Z -106.117,A -90.000,B 90.000,C 0.000} C_DIS
LIN {X 38.974,Y -46.256,Z -106.450,A -90.000,B 90.000,C 0.000} C_DIS
LIN {X 39.142,Y -46.236,Z -106.630,A -90.000,B 90.000,C 0.000} C_DIS
LIN {X 39.325,Y -46.213,Z -106.831,A -90.000,B 90.000,C 0.000} C_DIS
LIN {X 39.549,Y -46.177,Z -107.083,A -90.000,B 90.000,C 0.000} C_DIS
LIN {X 39.920,Y -46.125,Z -107.510,A -90.000,B 90.000,C 0.000} C_DIS
LIN {X 40.365,Y -46.048,Z -108.026,A -90.000,B 90.000,C 0.000} C_DIS
LIN {X 40.521,Y -46.017,Z -108.209,A -90.000,B 90.000,C 0.000} C_DIS
LIN {X 40.937,Y -45.934,Z -108.730,A -90.000,B 90.000,C 0.000} C_DIS
LIN {X 41.039,Y -45.914,Z -108.864,A -90.000,B 90.000,C 0.000} C_DIS
LIN {X 41.359,Y -45.863,Z -109.288,A -90.000,B 90.000,C 0.000} C_DIS
LIN {X 41.516,Y -45.838,Z -109.511,A -90.000,B 90.000,C 0.000} C_DIS
LIN {X 41.725,Y -45.800,Z -109.810,A -90.000,B 90.000,C 0.000} C_DIS
LIN {X 41.808,Y -45.784,Z -109.936,A -90.000,B 90.000,C 0.000} C_DIS
LIN {X 41.992,Y -45.731,Z -110.221,A -90.000,B 90.000,C 0.000} C_DIS
LIN {X 42.251,Y -45.655,Z -110.650,A -90.000,B 90.000,C 0.000} C_DIS
LIN {X 42.419,Y -45.605,Z -110.933,A -90.000,B 90.000,C 0.000} C_DIS
LIN {X 42.738,Y -45.510,Z -111.513,A -90.000,B 90.000,C 0.000} C_DIS
LIN {X 42.965,Y -45.441,Z -111.960,A -90.000,B 90.000,C 0.000} C_DIS
LIN {X 43.221,Y -45.363,Z -112.484,A -90.000,B 90.000,C 0.000} C_DIS
LIN {X 43.291,Y -45.341,Z -112.642,A -90.000,B 90.000,C 0.000} C_DIS
LIN {X 43.378,Y -45.308,Z -112.842,A -90.000,B 90.000,C 0.000} C_DIS
LIN {X 43.378,Y -60.000,Z -112.842,A -90.000,B 90.000,C 0.000} C_DIS
LIN {X -9.789,Y -60.000,Z -105.818,A -90.000,B 90.000,C 0.000} C_DIS
LIN {X -9.789,Y -45.308,Z -105.818,A -90.000,B 90.000,C 0.000} C_DIS
LIN {X -9.230,Y -45.397,Z -105.405,A -90.000,B 90.000,C 0.000} C_DIS
LIN {X -7.302,Y -45.690,Z -104.054,A -90.000,B 90.000,C 0.000} C_DIS
LIN {X -6.680,Y -45.784,Z -103.621,A -90.000,B 90.000,C 0.000} C_DIS
LIN {X -6.205,Y -45.854,Z -103.315,A -90.000,B 90.000,C 0.000} C_DIS
LIN {X -5.853,Y -45.904,Z -103.093,A -90.000,B 90.000,C 0.000} C_DIS
LIN {X -5.448,Y -45.960,Z -102.853,A -90.000,B 90.000,C 0.000} C_DIS
LIN {X -5.207,Y -45.998,Z -102.711,A -90.000,B 90.000,C 0.000} C_DIS
LIN {X -4.706,Y -46.076,Z -102.433,A -90.000,B 90.000,C 0.000} C_DIS
LIN {X -4.253,Y -46.145,Z -102.196,A -90.000,B 90.000,C 0.000} C_DIS
LIN {X -3.550,Y -46.252,Z -101.837,A -90.000,B 90.000,C 0.000} C_DIS
LIN {X -3.368,Y -46.276,Z -101.744,A -90.000,B 90.000,C 0.000} C_DIS
LIN {X -3.301,Y -46.283,Z -101.710,A -90.000,B 90.000,C 0.000} C_DIS
LIN {X -2.926,Y -46.330,Z -101.518,A -90.000,B 90.000,C 0.000} C_DIS
LIN {X -1.300,Y -46.498,Z -100.687,A -90.000,B 90.000,C 0.000} C_DIS
LIN {X -0.944,Y -46.539,Z -100.507,A -90.000,B 90.000,C 0.000} C_DIS
LIN {X -0.688,Y -46.565,Z -100.381,A -90.000,B 90.000,C 0.000} C_DIS
LIN {X -0.427,Y -46.590,Z -100.254,A -90.000,B 90.000,C 0.000} C_DIS
LIN {X -0.298,Y -46.601,Z -100.195,A -90.000,B 90.000,C 0.000} C_DIS
LIN {X 0.096,Y -46.620,Z -100.015,A -90.000,B 90.000,C 0.000} C_DIS
LIN {X 0.703,Y -46.648,Z -99.760,A -90.000,B 90.000,C 0.000} C_DIS
LIN {X 1.155,Y -46.669,Z -99.584,A -90.000,B 90.000,C 0.000} C_DIS
LIN {X 1.490,Y -46.690,Z -99.456,A -90.000,B 90.000,C 0.000} C_DIS
LIN {X 2.064,Y -46.727,Z -99.254,A -90.000,B 90.000,C 0.000} C_DIS
LIN {X 2.439,Y -46.751,Z -99.130,A -90.000,B 90.000,C 0.000} C_DIS
LIN {X 2.979,Y -46.786,Z -98.961,A -90.000,B 90.000,C 0.000} C_DIS
LIN {X 3.417,Y -46.803,Z -98.825,A -90.000,B 90.000,C 0.000} C_DIS
LIN {X 3.653,Y -46.805,Z -98.752,A -90.000,B 90.000,C 0.000} C_DIS
LIN {X 4.006,Y -46.801,Z -98.642,A -90.000,B 90.000,C 0.000} C_DIS
LIN {X 6.002,Y -46.746,Z -98.031,A -90.000,B 90.000,C 0.000} C_DIS
LIN {X 7.514,Y -46.723,Z -97.562,A -90.000,B 90.000,C 0.000} C_DIS
LIN {X 7.930,Y -46.716,Z -97.443,A -90.000,B 90.000,C 0.000} C_DIS
LIN {X 8.340,Y -46.692,Z -97.330,A -90.000,B 90.000,C 0.000} C_DIS
LIN {X 8.490,Y -46.684,Z -97.293,A -90.000,B 90.000,C 0.000} C_DIS
LIN {X 8.918,Y -46.655,Z -97.190,A -90.000,B 90.000,C 0.000} C_DIS
LIN {X 9.131,Y -46.637,Z -97.140,A -90.000,B 90.000,C 0.000} C_DIS
LIN {X 9.516,Y -46.607,Z -97.060,A -90.000,B 90.000,C 0.000} C_DIS
LIN {X 10.077,Y -46.566,Z -96.954,A -90.000,B 90.000,C 0.000} C_DIS
LIN {X 10.980,Y -46.505,Z -96.810,A -90.000,B 90.000,C 0.000} C_DIS
LIN {X 11.530,Y -46.478,Z -96.741,A -90.000,B 90.000,C 0.000} C_DIS
LIN {X 12.386,Y -46.441,Z -96.654,A -90.000,B 90.000,C 0.000} C_DIS
LIN {X 13.540,Y -46.380,Z -96.537,A -90.000,B 90.000,C 0.000} C_DIS
LIN {X 14.891,Y -46.325,Z -96.398,A -90.000,B 90.000,C 0.000} C_DIS
LIN {X 15.903,Y -46.284,Z -96.298,A -90.000,B 90.000,C 0.000} C_DIS
LIN {X 16.355,Y -46.257,Z -96.257,A -90.000,B 90.000,C 0.000} C_DIS
LIN {X 17.145,Y -46.220,Z -96.204,A -90.000,B 90.000,C 0.000} C_DIS
LIN {X 17.752,Y -46.196,Z -96.183,A -90.000,B 90.000,C 0.000} C_DIS
LIN {X 18.357,Y -46.177,Z -96.177,A -90.000,B 90.000,C 0.000} C_DIS
LIN {X 18.974,Y -46.165,Z -96.184,A -90.000,B 90.000,C 0.000} C_DIS
LIN {X 19.301,Y -46.160,Z -96.188,A -90.000,B 90.000,C 0.000} C_DIS
LIN {X 19.748,Y -46.154,Z -96.207,A -90.000,B 90.000,C 0.000} C_DIS
LIN {X 20.209,Y -46.150,Z -96.236,A -90.000,B 90.000,C 0.000} C_DIS
LIN {X 20.935,Y -46.147,Z -96.299,A -90.000,B 90.000,C 0.000} C_DIS
LIN {X 21.252,Y -46.148,Z -96.333,A -90.000,B 90.000,C 0.000} C_DIS
LIN {X 21.797,Y -46.153,Z -96.399,A -90.000,B 90.000,C 0.000} C_DIS
LIN {X 22.225,Y -46.162,Z -96.462,A -90.000,B 90.000,C 0.000} C_DIS
LIN {X 22.616,Y -46.170,Z -96.521,A -90.000,B 90.000,C 0.000} C_DIS
LIN {X 22.985,Y -46.180,Z -96.585,A -90.000,B 90.000,C 0.000} C_DIS
LIN {X 24.786,Y -46.193,Z -96.903,A -90.000,B 90.000,C 0.000} C_DIS
LIN {X 26.094,Y -46.210,Z -97.132,A -90.000,B 90.000,C 0.000} C_DIS
LIN {X 26.427,Y -46.216,Z -97.197,A -90.000,B 90.000,C 0.000} C_DIS
LIN {X 26.660,Y -46.216,Z -97.243,A -90.000,B 90.000,C 0.000} C_DIS
LIN {X 27.194,Y -46.210,Z -97.352,A -90.000,B 90.000,C 0.000} C_DIS
LIN {X 27.790,Y -46.206,Z -97.488,A -90.000,B 90.000,C 0.000} C_DIS
LIN {X 28.384,Y -46.208,Z -97.641,A -90.000,B 90.000,C 0.000} C_DIS
LIN {X 28.776,Y -46.212,Z -97.753,A -90.000,B 90.000,C 0.000} C_DIS
LIN {X 29.224,Y -46.219,Z -97.885,A -90.000,B 90.000,C 0.000} C_DIS
LIN {X 29.974,Y -46.238,Z -98.129,A -90.000,B 90.000,C 0.000} C_DIS
LIN {X 30.074,Y -46.241,Z -98.165,A -90.000,B 90.000,C 0.000} C_DIS
LIN {X 30.649,Y -46.239,Z -98.379,A -90.000,B 90.000,C 0.000} C_DIS
LIN {X 31.111,Y -46.239,Z -98.565,A -90.000,B 90.000,C 0.000} C_DIS
LIN {X 31.803,Y -46.241,Z -98.866,A -90.000,B 90.000,C 0.000} C_DIS
LIN {X 32.398,Y -46.246,Z -99.142,A -90.000,B 90.000,C 0.000} C_DIS
LIN {X 32.966,Y -46.257,Z -99.429,A -90.000,B 90.000,C 0.000} C_DIS
LIN {X 33.035,Y -46.258,Z -99.464,A -90.000,B 90.000,C 0.000} C_DIS
LIN {X 33.528,Y -46.259,Z -99.734,A -90.000,B 90.000,C 0.000} C_DIS
LIN {X 33.775,Y -46.256,Z -99.879,A -90.000,B 90.000,C 0.000} C_DIS
LIN {X 34.133,Y -46.243,Z -100.095,A -90.000,B 90.000,C 0.000} C_DIS
LIN {X 34.439,Y -46.234,Z -100.288,A -90.000,B 90.000,C 0.000} C_DIS
LIN {X 34.912,Y -46.222,Z -100.595,A -90.000,B 90.000,C 0.000} C_DIS
LIN {X 35.298,Y -46.213,Z -100.860,A -90.000,B 90.000,C 0.000} C_DIS
LIN {X 35.584,Y -46.208,Z -101.064,A -90.000,B 90.000,C 0.000} C_DIS
LIN {X 35.931,Y -46.204,Z -101.319,A -90.000,B 90.000,C 0.000} C_DIS
LIN {X 36.652,Y -46.199,Z -101.874,A -90.000,B 90.000,C 0.000} C_DIS
LIN {X 36.815,Y -46.197,Z -101.998,A -90.000,B 90.000,C 0.000} C_DIS
LIN {X 37.033,Y -46.187,Z -102.167,A -90.000,B 90.000,C 0.000} C_DIS
LIN {X 37.943,Y -46.131,Z -102.876,A -90.000,B 90.000,C 0.000} C_DIS
LIN {X 38.130,Y -46.118,Z -103.022,A -90.000,B 90.000,C 0.000} C_DIS
LIN {X 38.492,Y -46.096,Z -103.313,A -90.000,B 90.000,C 0.000} C_DIS
LIN {X 38.997,Y -46.067,Z -103.745,A -90.000,B 90.000,C 0.000} C_DIS
LIN {X 39.106,Y -46.059,Z -103.840,A -90.000,B 90.000,C 0.000} C_DIS
LIN {X 39.540,Y -46.027,Z -104.233,A -90.000,B 90.000,C 0.000} C_DIS
LIN {X 39.731,Y -46.010,Z -104.413,A -90.000,B 90.000,C 0.000} C_DIS
LIN {X 39.853,Y -45.996,Z -104.533,A -90.000,B 90.000,C 0.000} C_DIS
LIN {X 40.087,Y -45.966,Z -104.765,A -90.000,B 90.000,C 0.000} C_DIS
LIN {X 40.396,Y -45.916,Z -105.086,A -90.000,B 90.000,C 0.000} C_DIS
LIN {X 40.665,Y -45.873,Z -105.378,A -90.000,B 90.000,C 0.000} C_DIS
LIN {X 40.991,Y -45.821,Z -105.744,A -90.000,B 90.000,C 0.000} C_DIS
LIN {X 41.396,Y -45.758,Z -106.212,A -90.000,B 90.000,C 0.000} C_DIS
LIN {X 41.992,Y -45.673,Z -106.898,A -90.000,B 90.000,C 0.000} C_DIS
LIN {X 42.488,Y -45.605,Z -107.510,A -90.000,B 90.000,C 0.000} C_DIS
LIN {X 42.636,Y -45.585,Z -107.704,A -90.000,B 90.000,C 0.000} C_DIS
LIN {X 42.910,Y -45.519,Z -108.074,A -90.000,B 90.000,C 0.000} C_DIS
LIN {X 43.312,Y -45.420,Z -108.653,A -90.000,B 90.000,C 0.000} C_DIS
LIN {X 43.460,Y -45.384,Z -108.880,A -90.000,B 90.000,C 0.000} C_DIS
LIN {X 43.644,Y -45.329,Z -109.168,A -90.000,B 90.000,C 0.000} C_DIS
LIN {X 43.715,Y -45.308,Z -109.285,A -90.000,B 90.000,C 0.000} C_DIS
LIN {X 43.715,Y -60.000,Z -109.285,A -90.000,B 90.000,C 0.000} C_DIS
LIN {X -10.587,Y -60.000,Z -103.922,A -90.000,B 90.000,C 0.000} C_DIS
LIN {X -10.587,Y -45.308,Z -103.922,A -90.000,B 90.000,C 0.000} C_DIS
LIN {X -10.372,Y -45.344,Z -103.764,A -90.000,B 90.000,C 0.000} C_DIS
LIN {X -8.743,Y -45.611,Z -102.622,A -90.000,B 90.000,C 0.000} C_DIS
LIN {X -7.818,Y -45.745,Z -101.977,A -90.000,B 90.000,C 0.000} C_DIS
LIN {X -7.281,Y -45.821,Z -101.629,A -90.000,B 90.000,C 0.000} C_DIS
LIN {X -6.846,Y -45.883,Z -101.357,A -90.000,B 90.000,C 0.000} C_DIS
LIN {X -6.176,Y -45.987,Z -100.962,A -90.000,B 90.000,C 0.000} C_DIS
LIN {X -6.052,Y -46.004,Z -100.893,A -90.000,B 90.000,C 0.000} C_DIS
LIN {X -5.632,Y -46.049,Z -100.661,A -90.000,B 90.000,C 0.000} C_DIS
LIN {X -5.157,Y -46.100,Z -100.412,A -90.000,B 90.000,C 0.000} C_DIS
LIN {X -4.774,Y -46.141,Z -100.217,A -90.000,B 90.000,C 0.000} C_DIS
LIN {X -3.381,Y -46.325,Z -99.505,A -90.000,B 90.000,C 0.000} C_DIS
LIN {X -3.132,Y -46.354,Z -99.378,A -90.000,B 90.000,C 0.000} C_DIS
LIN {X -2.949,Y -46.371,Z -99.285,A -90.000,B 90.000,C 0.000} C_DIS
LIN {X -2.728,Y -46.386,Z -99.172,A -90.000,B 90.000,C 0.000} C_DIS
LIN {X -2.382,Y -46.405,Z -98.996,A -90.000,B 90.000,C 0.000} C_DIS
LIN {X -1.819,Y -46.447,Z -98.711,A -90.000,B 90.000,C 0.000} C_DIS
LIN {X -1.421,Y -46.478,Z -98.516,A -90.000,B 90.000,C 0.000} C_DIS
LIN {X -1.249,Y -46.488,Z -98.433,A -90.000,B 90.000,C 0.000} C_DIS
LIN {X -0.657,Y -46.522,Z -98.165,A -90.000,B 90.000,C 0.000} C_DIS
LIN {X -0.299,Y -46.540,Z -98.014,A -90.000,B 90.000,C 0.000} C_DIS
LIN {X -0.067,Y -46.550,Z -97.917,A -90.000,B 90.000,C 0.000} C_DIS
LIN {X 0.413,Y -46.564,Z -97.730,A -90.000,B 90.000,C 0.000} C_DIS
LIN {X 0.515,Y -46.565,Z -97.691,A -90.000,B 90.000,C 0.000} C_DIS
LIN {X 0.836,Y -46.559,Z -97.570,A -90.000,B 90.000,C 0.000} C_DIS
LIN {X 1.510,Y -46.550,Z -97.339,A -90.000,B 90.000,C 0.000} C_DIS
LIN {X 1.888,Y -46.546,Z -97.218,A -90.000,B 90.000,C 0.000} C_DIS
LIN {X 2.140,Y -46.544,Z -97.141,A -90.000,B 90.000,C 0.000} C_DIS
LIN {X 3.240,Y -46.545,Z -96.803,A -90.000,B 90.000,C 0.000} C_DIS
LIN {X 4.184,Y -46.546,Z -96.510,A -90.000,B 90.000,C 0.000} C_DIS
LIN {X 4.340,Y -46.544,Z -96.462,A -90.000,B 90.000,C 0.000} C_DIS
LIN {X 4.586,Y -46.536,Z -96.387,A -90.000,B 90.000,C 0.000} C_DIS
LIN {X 5.228,Y -46.496,Z -96.194,A -90.000,B 90.000,C 0.000} C_DIS
LIN {X 6.972,Y -46.341,Z -95.675,A -90.000,B 90.000,C 0.000} C_DIS
LIN {X 7.429,Y -46.304,Z -95.551,A -90.000,B 90.000,C 0.000} C_DIS
LIN {X 7.858,Y -46.272,Z -95.435,A -90.000,B 90.000,C 0.000} C_DIS
LIN {X 8.715,Y -46.214,Z -95.230,A -90.000,B 90.000,C 0.000} C_DIS
LIN {X 9.152,Y -46.187,Z -95.139,A -90.000,B 90.000,C 0.000} C_DIS
LIN {X 9.685,Y -46.149,Z -95.038,A -90.000,B 90.000,C 0.000} C_DIS
LIN {X 10.201,Y -46.120,Z -94.954,A -90.000,B 90.000,C 0.000} C_DIS
LIN {X 10.717,Y -46.076,Z -94.875,A -90.000,B 90.000,C 0.000} C_DIS
LIN {X 11.314,Y -46.030,Z -94.804,A -90.000,B 90.000,C 0.000} C_DIS
LIN {X 12.505,Y -45.943,Z -94.691,A -90.000,B 90.000,C 0.000} C_DIS
LIN {X 13.318,Y -45.888,Z -94.612,A -90.000,B 90.000,C 0.000} C_DIS
LIN {X 14.749,Y -45.787,Z -94.476,A -90.000,B 90.000,C 0.000} C_DIS
LIN {X 16.148,Y -45.706,Z -94.345,A -90.000,B 90.000,C 0.000} C_DIS
LIN {X 17.058,Y -45.663,Z -94.285,A -90.000,B 90.000,C 0.000} C_DIS
LIN {X 17.714,Y -45.643,Z -94.262,A -90.000,B 90.000,C 0.000} C_DIS
LIN {X 18.367,Y -45.628,Z -94.254,A -90.000,B 90.000,C 0.000} C_DIS
LIN {X 19.328,Y -45.610,Z -94.266,A -90.000,B 90.000,C 0.000} C_DIS
LIN {X 19.864,Y -45.604,Z -94.288,A -90.000,B 90.000,C 0.000} C_DIS
LIN {X 20.373,Y -45.601,Z -94.320,A -90.000,B 90.000,C 0.000} C_DIS
LIN {X 21.142,Y -45.601,Z -94.386,A -90.000,B 90.000,C 0.000} C_DIS
LIN {X 21.488,Y -45.603,Z -94.423,A -90.000,B 90.000,C 0.000} C_DIS
LIN {X 22.088,Y -45.608,Z -94.497,A -90.000,B 90.000,C 0.000} C_DIS
LIN {X 22.956,Y -45.623,Z -94.628,A -90.000,B 90.000,C 0.000} C_DIS
LIN {X 23.483,Y -45.637,Z -94.718,A -90.000,B 90.000,C 0.000} C_DIS
LIN {X 26.471,Y -45.677,Z -95.242,A -90.000,B 90.000,C 0.000} C_DIS
LIN {X 26.997,Y -45.688,Z -95.344,A -90.000,B 90.000,C 0.000} C_DIS
LIN {X 27.549,Y -45.687,Z -95.455,A -90.000,B 90.000,C 0.000} C_DIS
LIN {X 28.275,Y -45.689,Z -95.618,A -90.000,B 90.000,C 0.000} C_DIS
LIN {X 28.914,Y -45.697,Z -95.782,A -90.000,B 90.000,C 0.000} C_DIS
LIN {X 29.331,Y -45.705,Z -95.899,A -90.000,B 90.000,C 0.000} C_DIS
LIN {X 29.836,Y -45.717,Z -96.048,A -90.000,B 90.000,C 0.000} C_DIS
LIN {X 30.640,Y -45.743,Z -96.310,A -90.000,B 90.000,C 0.000} C_DIS
LIN {X 30.740,Y -45.745,Z -96.346,A -90.000,B 90.000,C 0.000} C_DIS
LIN {X 31.370,Y -45.743,Z -96.580,A -90.000,B 90.000,C 0.000} C_DIS
LIN {X 31.888,Y -45.746,Z -96.789,A -90.000,B 90.000,C 0.000} C_DIS
LIN {X 32.620,Y -45.755,Z -97.107,A -90.000,B 90.000,C 0.000} C_DIS
LIN {X 33.171,Y -45.765,Z -97.361,A -90.000,B 90.000,C 0.000} C_DIS
LIN {X 33.281,Y -45.766,Z -97.413,A -90.000,B 90.000,C 0.000} C_DIS
LIN {X 33.969,Y -45.779,Z -97.762,A -90.000,B 90.000,C 0.000} C_DIS
LIN {X 34.222,Y -45.785,Z -97.899,A -90.000,B 90.000,C 0.000} C_DIS
LIN {X 34.503,Y -45.784,Z -98.054,A -90.000,B 90.000,C 0.000} C_DIS
LIN {X 34.935,Y -45.785,Z -98.307,A -90.000,B 90.000,C 0.000} C_DIS
LIN {X 35.160,Y -45.786,Z -98.441,A -90.000,B 90.000,C 0.000} C_DIS
LIN {X 35.436,Y -45.788,Z -98.612,A -90.000,B 90.000,C 0.000} C_DIS
LIN {X 36.009,Y -45.787,Z -98.980,A -90.000,B 90.000,C 0.000} C_DIS
LIN {X 36.429,Y -45.790,Z -99.265,A -90.000,B 90.000,C 0.000} C_DIS
LIN {X 36.809,Y -45.795,Z -99.536,A -90.000,B 90.000,C 0.000} C_DIS
LIN {X 37.123,Y -45.800,Z -99.765,A -90.000,B 90.000,C 0.000} C_DIS
LIN {X 37.339,Y -45.805,Z -99.929,A -90.000,B 90.000,C 0.000} C_DIS
LIN {X 37.566,Y -45.807,Z -100.103,A -90.000,B 90.000,C 0.000} C_DIS
LIN {X 38.002,Y -45.785,Z -100.443,A -90.000,B 90.000,C 0.000} C_DIS
LIN {X 39.340,Y -45.704,Z -101.485,A -90.000,B 90.000,C 0.000} C_DIS
LIN {X 39.749,Y -45.680,Z -101.814,A -90.000,B 90.000,C 0.000} C_DIS
LIN {X 40.403,Y -45.645,Z -102.375,A -90.000,B 90.000,C 0.000} C_DIS
LIN {X 40.606,Y -45.635,Z -102.557,A -90.000,B 90.000,C 0.000} C_DIS
LIN {X 40.861,Y -45.609,Z -102.790,A -90.000,B 90.000,C 0.000} C_DIS
LIN {X 41.073,Y -45.587,Z -102.991,A -90.000,B 90.000,C 0.000} C_DIS
LIN {X 41.463,Y -45.548,Z -103.374,A -90.000,B 90.000,C 0.000} C_DIS
LIN {X 41.809,Y -45.510,Z -103.729,A -90.000,B 90.000,C 0.000} C_DIS
LIN {X 42.129,Y -45.476,Z -104.074,A -90.000,B 90.000,C 0.000} C_DIS
LIN {X 42.489,Y -45.438,Z -104.474,A -90.000,B 90.000,C 0.000} C_DIS
LIN {X 42.718,Y -45.415,Z -104.735,A -90.000,B 90.000,C 0.000} C_DIS
LIN {X 42.945,Y -45.385,Z -104.996,A -90.000,B 90.000,C 0.000} C_DIS
LIN {X 43.325,Y -45.326,Z -105.435,A -90.000,B 90.000,C 0.000} C_DIS
LIN {X 43.450,Y -45.308,Z -105.579,A -90.000,B 90.000,C 0.000} C_DIS
LIN {X 43.450,Y -60.000,Z -105.579,A -90.000,B 90.000,C 0.000} C_DIS
LIN {X 37.100,Y -60.000,Z -97.374,A -90.000,B 90.000,C 0.000} C_DIS
LIN {X 37.100,Y -45.308,Z -97.374,A -90.000,B 90.000,C 0.000} C_DIS
LIN {X 37.355,Y -45.314,Z -97.546,A -90.000,B 90.000,C 0.000} C_DIS
LIN {X 37.607,Y -45.316,Z -97.719,A -90.000,B 90.000,C 0.000} C_DIS
LIN {X 38.078,Y -45.321,Z -98.057,A -90.000,B 90.000,C 0.000} C_DIS
LIN {X 38.273,Y -45.320,Z -98.200,A -90.000,B 90.000,C 0.000} C_DIS
LIN {X 39.169,Y -45.308,Z -98.889,A -90.000,B 90.000,C 0.000} C_DIS
LIN {X 39.169,Y -60.000,Z -98.889,A -90.000,B 90.000,C 0.000} C_DIS
LIN {X -11.226,Y -60.000,Z -101.922,A -90.000,B 90.000,C 0.000} C_DIS
LIN {X -11.226,Y -45.308,Z -101.922,A -90.000,B 90.000,C 0.000} C_DIS
LIN {X -10.946,Y -45.353,Z -101.726,A -90.000,B 90.000,C 0.000} C_DIS
LIN {X -10.061,Y -45.473,Z -101.107,A -90.000,B 90.000,C 0.000} C_DIS
LIN {X -8.895,Y -45.666,Z -100.294,A -90.000,B 90.000,C 0.000} C_DIS
LIN {X -8.560,Y -45.721,Z -100.077,A -90.000,B 90.000,C 0.000} C_DIS
LIN {X -8.379,Y -45.746,Z -99.960,A -90.000,B 90.000,C 0.000} C_DIS
LIN {X -8.028,Y -45.783,Z -99.739,A -90.000,B 90.000,C 0.000} C_DIS
LIN {X -7.856,Y -45.805,Z -99.632,A -90.000,B 90.000,C 0.000} C_DIS
LIN {X -7.137,Y -45.900,Z -99.210,A -90.000,B 90.000,C 0.000} C_DIS
LIN {X -6.951,Y -45.923,Z -99.107,A -90.000,B 90.000,C 0.000} C_DIS
LIN {X -6.519,Y -45.969,Z -98.870,A -90.000,B 90.000,C 0.000} C_DIS
LIN {X -6.245,Y -45.999,Z -98.726,A -90.000,B 90.000,C 0.000} C_DIS
LIN {X -6.025,Y -46.027,Z -98.611,A -90.000,B 90.000,C 0.000} C_DIS
LIN {X -5.803,Y -46.053,Z -98.498,A -90.000,B 90.000,C 0.000} C_DIS
LIN {X -5.570,Y -46.073,Z -98.380,A -90.000,B 90.000,C 0.000} C_DIS
LIN {X -5.393,Y -46.086,Z -98.290,A -90.000,B 90.000,C 0.000} C_DIS
LIN {X -3.824,Y -46.171,Z -97.497,A -90.000,B 90.000,C 0.000} C_DIS
LIN {X -2.797,Y -46.248,Z -96.975,A -90.000,B 90.000,C 0.000} C_DIS
LIN {X -2.682,Y -46.257,Z -96.917,A -90.000,B 90.000,C 0.000} C_DIS
LIN {X -2.497,Y -46.265,Z -96.827,A -90.000,B 90.000,C 0.000} C_DIS
LIN {X -2.280,Y -46.267,Z -96.723,A -90.000,B 90.000,C 0.000} C_DIS
LIN {X -2.059,Y -46.265,Z -96.618,A -90.000,B 90.000,C 0.000} C_DIS
LIN {X -1.467,Y -46.262,Z -96.355,A -90.000,B 90.000,C 0.000} C_DIS
LIN {X -0.777,Y -46.266,Z -96.069,A -90.000,B 90.000,C 0.000} C_DIS
LIN {X 0.099,Y -46.276,Z -95.733,A -90.000,B 90.000,C 0.000} C_DIS
LIN {X 0.179,Y -46.277,Z -95.703,A -90.000,B 90.000,C 0.000} C_DIS
LIN {X 0.306,Y -46.279,Z -95.658,A -90.000,B 90.000,C 0.000} C_DIS
LIN {X 0.765,Y -46.273,Z -95.501,A -90.000,B 90.000,C 0.000} C_DIS
LIN {X 0.910,Y -46.273,Z -95.452,A -90.000,B 90.000,C 0.000} C_DIS
LIN {X 1.047,Y -46.271,Z -95.408,A -90.000,B 90.000,C 0.000} C_DIS
LIN {X 1.387,Y -46.259,Z -95.301,A -90.000,B 90.000,C 0.000} C_DIS
LIN {X 1.771,Y -46.246,Z -95.186,A -90.000,B 90.000,C 0.000} C_DIS
LIN {X 4.002,Y -46.094,Z -94.526,A -90.000,B 90.000,C 0.000} C_DIS
LIN {X 5.577,Y -45.984,Z -94.052,A -90.000,B 90.000,C 0.000} C_DIS
LIN {X 5.941,Y -45.952,Z -93.944,A -90.000,B 90.000,C 0.000} C_DIS
LIN {X 6.245,Y -45.927,Z -93.853,A -90.000,B 90.000,C 0.000} C_DIS
LIN {X 6.429,Y -45.905,Z -93.800,A -90.000,B 90.000,C 0.000} C_DIS
LIN {X 7.162,Y -45.824,Z -93.607,A -90.000,B 90.000,C 0.000} C_DIS
LIN {X 7.377,Y -45.799,Z -93.552,A -90.000,B 90.000,C 0.000} C_DIS
LIN {X 8.289,Y -45.700,Z -93.345,A -90.000,B 90.000,C 0.000} C_DIS
LIN {X 8.801,Y -45.650,Z -93.244,A -90.000,B 90.000,C 0.000} C_DIS
LIN {X 9.344,Y -45.601,Z -93.145,A -90.000,B 90.000,C 0.000} C_DIS
LIN {X 9.826,Y -45.561,Z -93.070,A -90.000,B 90.000,C 0.000} C_DIS
LIN {X 10.439,Y -45.505,Z -92.978,A -90.000,B 90.000,C 0.000} C_DIS
LIN {X 11.101,Y -45.452,Z -92.901,A -90.000,B 90.000,C 0.000} C_DIS
LIN {X 13.309,Y -45.308,Z -92.686,A -90.000,B 90.000,C 0.000} C_DIS
LIN {X 13.309,Y -60.000,Z -92.686,A -90.000,B 90.000,C 0.000} C_DIS
LIN {X -11.534,Y -60.000,Z -99.701,A -90.000,B 90.000,C 0.000} C_DIS
LIN {X -11.534,Y -45.308,Z -99.701,A -90.000,B 90.000,C 0.000} C_DIS
LIN {X -11.421,Y -45.324,Z -99.622,A -90.000,B 90.000,C 0.000} C_DIS
LIN {X -10.873,Y -45.413,Z -99.239,A -90.000,B 90.000,C 0.000} C_DIS
LIN {X -10.707,Y -45.435,Z -99.124,A -90.000,B 90.000,C 0.000} C_DIS
LIN {X -9.961,Y -45.508,Z -98.609,A -90.000,B 90.000,C 0.000} C_DIS
LIN {X -9.410,Y -45.562,Z -98.256,A -90.000,B 90.000,C 0.000} C_DIS
LIN {X -8.929,Y -45.625,Z -97.954,A -90.000,B 90.000,C 0.000} C_DIS
LIN {X -8.801,Y -45.642,Z -97.876,A -90.000,B 90.000,C 0.000} C_DIS
LIN {X -8.252,Y -45.713,Z -97.554,A -90.000,B 90.000,C 0.000} C_DIS
LIN {X -8.150,Y -45.724,Z -97.495,A -90.000,B 90.000,C 0.000} C_DIS
LIN {X -7.967,Y -45.740,Z -97.392,A -90.000,B 90.000,C 0.000} C_DIS
LIN {X -7.465,Y -45.767,Z -97.119,A -90.000,B 90.000,C 0.000} C_DIS
LIN {X -7.187,Y -45.784,Z -96.974,A -90.000,B 90.000,C 0.000} C_DIS
LIN {X -6.944,Y -45.803,Z -96.849,A -90.000,B 90.000,C 0.000} C_DIS
LIN {X -5.294,Y -45.932,Z -96.011,A -90.000,B 90.000,C 0.000} C_DIS
LIN {X -5.096,Y -45.944,Z -95.911,A -90.000,B 90.000,C 0.000} C_DIS
LIN {X -4.928,Y -45.945,Z -95.827,A -90.000,B 90.000,C 0.000} C_DIS
LIN {X -3.531,Y -45.927,Z -95.136,A -90.000,B 90.000,C 0.000} C_DIS
LIN {X -2.861,Y -45.921,Z -94.819,A -90.000,B 90.000,C 0.000} C_DIS
LIN {X -2.221,Y -45.922,Z -94.534,A -90.000,B 90.000,C 0.000} C_DIS
LIN {X -1.941,Y -45.923,Z -94.418,A -90.000,B 90.000,C 0.000} C_DIS
LIN {X -1.479,Y -45.919,Z -94.229,A -90.000,B 90.000,C 0.000} C_DIS
LIN {X -1.404,Y -45.918,Z -94.200,A -90.000,B 90.000,C 0.000} C_DIS
LIN {X -1.219,Y -45.912,Z -94.131,A -90.000,B 90.000,C 0.000} C_DIS
LIN {X -0.539,Y -45.876,Z -93.879,A -90.000,B 90.000,C 0.000} C_DIS
LIN {X -0.330,Y -45.866,Z -93.808,A -90.000,B 90.000,C 0.000} C_DIS
LIN {X 0.252,Y -45.834,Z -93.615,A -90.000,B 90.000,C 0.000} C_DIS
LIN {X 0.842,Y -45.804,Z -93.431,A -90.000,B 90.000,C 0.000} C_DIS
LIN {X 1.271,Y -45.783,Z -93.304,A -90.000,B 90.000,C 0.000} C_DIS
LIN {X 3.006,Y -45.664,Z -92.791,A -90.000,B 90.000,C 0.000} C_DIS
LIN {X 3.683,Y -45.596,Z -92.595,A -90.000,B 90.000,C 0.000} C_DIS
LIN {X 5.166,Y -45.431,Z -92.165,A -90.000,B 90.000,C 0.000} C_DIS
LIN {X 5.882,Y -45.347,Z -91.959,A -90.000,B 90.000,C 0.000} C_DIS
LIN {X 6.235,Y -45.308,Z -91.866,A -90.000,B 90.000,C 0.000} C_DIS
LIN {X 6.235,Y -60.000,Z -91.866,A -90.000,B 90.000,C 0.000} C_DIS
LIN {X -11.138,Y -60.000,Z -97.002,A -90.000,B 90.000,C 0.000} C_DIS
LIN {X -11.138,Y -45.308,Z -97.002,A -90.000,B 90.000,C 0.000} C_DIS
LIN {X -11.023,Y -45.320,Z -96.924,A -90.000,B 90.000,C 0.000} C_DIS
LIN {X -10.763,Y -45.346,Z -96.758,A -90.000,B 90.000,C 0.000} C_DIS
LIN {X -10.568,Y -45.368,Z -96.632,A -90.000,B 90.000,C 0.000} C_DIS
LIN {X -10.391,Y -45.383,Z -96.521,A -90.000,B 90.000,C 0.000} C_DIS
LIN {X -9.940,Y -45.403,Z -96.243,A -90.000,B 90.000,C 0.000} C_DIS
LIN {X -9.784,Y -45.411,Z -96.150,A -90.000,B 90.000,C 0.000} C_DIS
LIN {X -9.098,Y -45.446,Z -95.756,A -90.000,B 90.000,C 0.000} C_DIS
LIN {X -8.592,Y -45.473,Z -95.478,A -90.000,B 90.000,C 0.000} C_DIS
LIN {X -8.302,Y -45.494,Z -95.322,A -90.000,B 90.000,C 0.000} C_DIS
LIN {X -7.785,Y -45.535,Z -95.054,A -90.000,B 90.000,C 0.000} C_DIS
LIN {X -7.586,Y -45.546,Z -94.954,A -90.000,B 90.000,C 0.000} C_DIS
LIN {X -7.151,Y -45.554,Z -94.737,A -90.000,B 90.000,C 0.000} C_DIS
LIN {X -5.671,Y -45.561,Z -94.004,A -90.000,B 90.000,C 0.000} C_DIS
LIN {X -4.379,Y -45.568,Z -93.361,A -90.000,B 90.000,C 0.000} C_DIS
LIN {X -4.050,Y -45.569,Z -93.204,A -90.000,B 90.000,C 0.000} C_DIS
LIN {X -3.660,Y -45.546,Z -93.024,A -90.000,B 90.000,C 0.000} C_DIS
LIN {X -2.968,Y -45.500,Z -92.728,A -90.000,B 90.000,C 0.000} C_DIS
LIN {X -2.173,Y -45.451,Z -92.412,A -90.000,B 90.000,C 0.000} C_DIS
LIN {X -1.439,Y -45.412,Z -92.141,A -90.000,B 90.000,C 0.000} C_DIS
LIN {X -1.189,Y -45.396,Z -92.050,A -90.000,B 90.000,C 0.000} C_DIS
LIN {X -0.572,Y -45.360,Z -91.844,A -90.000,B 90.000,C 0.000} C_DIS
LIN {X -0.346,Y -45.347,Z -91.769,A -90.000,B 90.000,C 0.000} C_DIS
LIN {X -0.158,Y -45.337,Z -91.711,A -90.000,B 90.000,C 0.000} C_DIS
LIN {X 0.212,Y -45.308,Z -91.599,A -90.000,B 90.000,C 0.000} C_DIS
LIN {X 0.804,Y -45.308,Z -91.576,A -90.000,B 90.000,C 0.000} C_DIS
LIN {X 1.493,Y -45.308,Z -91.560,A -90.000,B 90.000,C 0.000} C_DIS
LIN {X 1.924,Y -45.308,Z -91.574,A -90.000,B 90.000,C 0.000} C_DIS
LIN {X 4.515,Y -45.308,Z -91.734,A -90.000,B 90.000,C 0.000} C_DIS
LIN {X 4.796,Y -45.308,Z -91.752,A -90.000,B 90.000,C 0.000} C_DIS
LIN {X 6.356,Y -45.308,Z -91.875,A -90.000,B 90.000,C 0.000} C_DIS
LIN {X 7.774,Y -45.308,Z -92.041,A -90.000,B 90.000,C 0.000} C_DIS
LIN {X 10.035,Y -45.308,Z -92.284,A -90.000,B 90.000,C 0.000} C_DIS
LIN {X 10.691,Y -45.308,Z -92.378,A -90.000,B 90.000,C 0.000} C_DIS
LIN {X 13.512,Y -45.308,Z -92.710,A -90.000,B 90.000,C 0.000} C_DIS
LIN {X 14.170,Y -45.308,Z -92.782,A -90.000,B 90.000,C 0.000} C_DIS
LIN {X 16.495,Y -45.308,Z -93.091,A -90.000,B 90.000,C 0.000} C_DIS
LIN {X 19.406,Y -45.308,Z -93.388,A -90.000,B 90.000,C 0.000} C_DIS
LIN {X 20.207,Y -45.308,Z -93.443,A -90.000,B 90.000,C 0.000} C_DIS
LIN {X 22.398,Y -45.308,Z -93.665,A -90.000,B 90.000,C 0.000} C_DIS
LIN {X 23.711,Y -45.308,Z -93.751,A -90.000,B 90.000,C 0.000} C_DIS
LIN {X 25.625,Y -45.308,Z -94.009,A -90.000,B 90.000,C 0.000} C_DIS
LIN {X 27.290,Y -45.308,Z -94.170,A -90.000,B 90.000,C 0.000} C_DIS
LIN {X 29.336,Y -45.308,Z -94.598,A -90.000,B 90.000,C 0.000} C_DIS
LIN {X 30.870,Y -45.308,Z -94.859,A -90.000,B 90.000,C 0.000} C_DIS
LIN {X 31.103,Y -45.308,Z -94.908,A -90.000,B 90.000,C 0.000} C_DIS
LIN {X 32.548,Y -45.308,Z -95.321,A -90.000,B 90.000,C 0.000} C_DIS
LIN {X 34.596,Y -45.308,Z -96.049,A -90.000,B 90.000,C 0.000} C_DIS
LIN {X 35.269,Y -45.308,Z -96.346,A -90.000,B 90.000,C 0.000} C_DIS
LIN {X 36.135,Y -45.308,Z -96.818,A -90.000,B 90.000,C 0.000} C_DIS
LIN {X 37.355,Y -45.308,Z -97.521,A -90.000,B 90.000,C 0.000} C_DIS
LIN {X 38.030,Y -45.308,Z -97.958,A -90.000,B 90.000,C 0.000} C_DIS
LIN {X 38.222,Y -45.308,Z -98.096,A -90.000,B 90.000,C 0.000} C_DIS
LIN {X 39.366,Y -45.308,Z -99.055,A -90.000,B 90.000,C 0.000} C_DIS
LIN {X 40.967,Y -45.308,Z -100.618,A -90.000,B 90.000,C 0.000} C_DIS
LIN {X 41.126,Y -45.308,Z -100.793,A -90.000,B 90.000,C 0.000} C_DIS
LIN {X 41.215,Y -45.308,Z -100.903,A -90.000,B 90.000,C 0.000} C_DIS
LIN {X 41.334,Y -45.308,Z -101.108,A -90.000,B 90.000,C 0.000} C_DIS
LIN {X 42.351,Y -45.308,Z -102.962,A -90.000,B 90.000,C 0.000} C_DIS
LIN {X 43.259,Y -45.308,Z -104.862,A -90.000,B 90.000,C 0.000} C_DIS
LIN {X 43.333,Y -45.308,Z -105.087,A -90.000,B 90.000,C 0.000} C_DIS
LIN {X 43.372,Y -45.308,Z -105.280,A -90.000,B 90.000,C 0.000} C_DIS
LIN {X 43.457,Y -45.308,Z -105.604,A -90.000,B 90.000,C 0.000} C_DIS
LIN {X 43.482,Y -45.308,Z -105.839,A -90.000,B 90.000,C 0.000} C_DIS
LIN {X 43.740,Y -45.308,Z -108.978,A -90.000,B 90.000,C 0.000} C_DIS
LIN {X 43.509,Y -45.308,Z -111.746,A -90.000,B 90.000,C 0.000} C_DIS
LIN {X 43.414,Y -45.308,Z -112.695,A -90.000,B 90.000,C 0.000} C_DIS
LIN {X 42.909,Y -45.308,Z -114.801,A -90.000,B 90.000,C 0.000} C_DIS
LIN {X 42.510,Y -45.308,Z -116.194,A -90.000,B 90.000,C 0.000} C_DIS
LIN {X 42.452,Y -45.308,Z -116.356,A -90.000,B 90.000,C 0.000} C_DIS
LIN {X 41.931,Y -45.308,Z -117.489,A -90.000,B 90.000,C 0.000} C_DIS
LIN {X 40.948,Y -45.308,Z -119.574,A -90.000,B 90.000,C 0.000} C_DIS
LIN {X 40.807,Y -45.308,Z -119.818,A -90.000,B 90.000,C 0.000} C_DIS
LIN {X 39.303,Y -45.308,Z -122.150,A -90.000,B 90.000,C 0.000} C_DIS
LIN {X 38.803,Y -45.308,Z -122.863,A -90.000,B 90.000,C 0.000} C_DIS
LIN {X 37.272,Y -45.308,Z -124.793,A -90.000,B 90.000,C 0.000} C_DIS
LIN {X 37.090,Y -45.308,Z -125.008,A -90.000,B 90.000,C 0.000} C_DIS
LIN {X 34.745,Y -45.308,Z -127.609,A -90.000,B 90.000,C 0.000} C_DIS
LIN {X 33.643,Y -45.308,Z -128.664,A -90.000,B 90.000,C 0.000} C_DIS
LIN {X 32.208,Y -45.308,Z -130.152,A -90.000,B 90.000,C 0.000} C_DIS
LIN {X 31.647,Y -45.308,Z -130.729,A -90.000,B 90.000,C 0.000} C_DIS
LIN {X 30.340,Y -45.308,Z -131.894,A -90.000,B 90.000,C 0.000} C_DIS
LIN {X 28.420,Y -45.308,Z -133.853,A -90.000,B 90.000,C 0.000} C_DIS
LIN {X 28.085,Y -45.308,Z -134.135,A -90.000,B 90.000,C 0.000} C_DIS
LIN {X 25.749,Y -45.308,Z -136.318,A -90.000,B 90.000,C 0.000} C_DIS
LIN {X 25.499,Y -45.308,Z -136.497,A -90.000,B 90.000,C 0.000} C_DIS
LIN {X 23.270,Y -45.308,Z -138.216,A -90.000,B 90.000,C 0.000} C_DIS
LIN {X 22.984,Y -45.308,Z -138.420,A -90.000,B 90.000,C 0.000} C_DIS
LIN {X 22.646,Y -45.308,Z -138.611,A -90.000,B 90.000,C 0.000} C_DIS
LIN {X 20.374,Y -45.308,Z -139.943,A -90.000,B 90.000,C 0.000} C_DIS
LIN {X 20.062,Y -45.308,Z -140.105,A -90.000,B 90.000,C 0.000} C_DIS
LIN {X 16.943,Y -45.308,Z -141.374,A -90.000,B 90.000,C 0.000} C_DIS
LIN {X 16.611,Y -45.308,Z -141.490,A -90.000,B 90.000,C 0.000} C_DIS
LIN {X 13.243,Y -45.308,Z -142.403,A -90.000,B 90.000,C 0.000} C_DIS
LIN {X 12.823,Y -45.308,Z -142.511,A -90.000,B 90.000,C 0.000} C_DIS
LIN {X 12.478,Y -45.308,Z -142.579,A -90.000,B 90.000,C 0.000} C_DIS
LIN {X 11.546,Y -45.308,Z -142.713,A -90.000,B 90.000,C 0.000} C_DIS
LIN {X 8.355,Y -45.308,Z -143.108,A -90.000,B 90.000,C 0.000} C_DIS
LIN {X 8.004,Y -45.308,Z -143.126,A -90.000,B 90.000,C 0.000} C_DIS
LIN {X 6.839,Y -45.308,Z -143.151,A -90.000,B 90.000,C 0.000} C_DIS
LIN {X 3.906,Y -45.308,Z -143.121,A -90.000,B 90.000,C 0.000} C_DIS
LIN {X 3.556,Y -45.308,Z -143.090,A -90.000,B 90.000,C 0.000} C_DIS
LIN {X 1.922,Y -45.308,Z -142.775,A -90.000,B 90.000,C 0.000} C_DIS
LIN {X -0.413,Y -45.308,Z -142.435,A -90.000,B 90.000,C 0.000} C_DIS
LIN {X -0.722,Y -45.308,Z -142.355,A -90.000,B 90.000,C 0.000} C_DIS
LIN {X -2.333,Y -45.308,Z -141.699,A -90.000,B 90.000,C 0.000} C_DIS
LIN {X -4.118,Y -45.308,Z -141.063,A -90.000,B 90.000,C 0.000} C_DIS
LIN {X -4.411,Y -45.308,Z -140.936,A -90.000,B 90.000,C 0.000} C_DIS
LIN {X -4.680,Y -45.308,Z -140.764,A -90.000,B 90.000,C 0.000} C_DIS
LIN {X -6.700,Y -45.308,Z -139.376,A -90.000,B 90.000,C 0.000} C_DIS
LIN {X -7.520,Y -45.308,Z -138.859,A -90.000,B 90.000,C 0.000} C_DIS
LIN {X -7.731,Y -45.308,Z -138.672,A -90.000,B 90.000,C 0.000} C_DIS
LIN {X -8.765,Y -45.308,Z -137.539,A -90.000,B 90.000,C 0.000} C_DIS
LIN {X -8.940,Y -45.308,Z -137.317,A -90.000,B 90.000,C 0.000} C_DIS
LIN {X -9.320,Y -45.308,Z -136.747,A -90.000,B 90.000,C 0.000} C_DIS
LIN {X -9.355,Y -45.308,Z -136.691,A -90.000,B 90.000,C 0.000} C_DIS
LIN {X -9.938,Y -45.308,Z -135.722,A -90.000,B 90.000,C 0.000} C_DIS
LIN {X -10.043,Y -45.308,Z -135.454,A -90.000,B 90.000,C 0.000} C_DIS
LIN {X -10.437,Y -45.308,Z -134.320,A -90.000,B 90.000,C 0.000} C_DIS
LIN {X -10.524,Y -45.308,Z -134.052,A -90.000,B 90.000,C 0.000} C_DIS
LIN {X -10.535,Y -45.308,Z -134.008,A -90.000,B 90.000,C 0.000} C_DIS
LIN {X -10.787,Y -45.308,Z -132.485,A -90.000,B 90.000,C 0.000} C_DIS
LIN {X -10.817,Y -45.308,Z -132.250,A -90.000,B 90.000,C 0.000} C_DIS
LIN {X -10.823,Y -45.308,Z -131.950,A -90.000,B 90.000,C 0.000} C_DIS
LIN {X -10.772,Y -45.308,Z -131.326,A -90.000,B 90.000,C 0.000} C_DIS
LIN {X -10.600,Y -45.308,Z -129.677,A -90.000,B 90.000,C 0.000} C_DIS
LIN {X -10.409,Y -45.308,Z -128.611,A -90.000,B 90.000,C 0.000} C_DIS
LIN {X -10.340,Y -45.308,Z -128.385,A -90.000,B 90.000,C 0.000} C_DIS
LIN {X -10.040,Y -45.308,Z -127.470,A -90.000,B 90.000,C 0.000} C_DIS
LIN {X -9.489,Y -45.308,Z -125.451,A -90.000,B 90.000,C 0.000} C_DIS
LIN {X -9.420,Y -45.308,Z -125.225,A -90.000,B 90.000,C 0.000} C_DIS
LIN {X -9.401,Y -45.308,Z -125.186,A -90.000,B 90.000,C 0.000} C_DIS
LIN {X -9.362,Y -45.308,Z -125.067,A -90.000,B 90.000,C 0.000} C_DIS
LIN {X -8.618,Y -45.308,Z -122.923,A -90.000,B 90.000,C 0.000} C_DIS
LIN {X -8.501,Y -45.308,Z -122.280,A -90.000,B 90.000,C 0.000} C_DIS
LIN {X -8.432,Y -45.308,Z -122.053,A -90.000,B 90.000,C 0.000} C_DIS
LIN {X -7.787,Y -45.308,Z -120.416,A -90.000,B 90.000,C 0.000} C_DIS
LIN {X -7.574,Y -45.308,Z -119.006,A -90.000,B 90.000,C 0.000} C_DIS
LIN {X -7.532,Y -45.308,Z -118.815,A -90.000,B 90.000,C 0.000} C_DIS
LIN {X -7.289,Y -45.308,Z -118.218,A -90.000,B 90.000,C 0.000} C_DIS
LIN {X -7.153,Y -45.308,Z -116.647,A -90.000,B 90.000,C 0.000} C_DIS
LIN {X -7.061,Y -45.308,Z -115.931,A -90.000,B 90.000,C 0.000} C_DIS
LIN {X -7.085,Y -45.308,Z -115.774,A -90.000,B 90.000,C 0.000} C_DIS
LIN {X -7.095,Y -45.308,Z -115.595,A -90.000,B 90.000,C 0.000} C_DIS
LIN {X -6.982,Y -45.308,Z -113.494,A -90.000,B 90.000,C 0.000} C_DIS
LIN {X -7.376,Y -45.308,Z -112.098,A -90.000,B 90.000,C 0.000} C_DIS
LIN {X -7.438,Y -45.308,Z -111.311,A -90.000,B 90.000,C 0.000} C_DIS
LIN {X -7.863,Y -45.308,Z -110.395,A -90.000,B 90.000,C 0.000} C_DIS
LIN {X -7.921,Y -45.308,Z -110.230,A -90.000,B 90.000,C 0.000} C_DIS
LIN {X -8.239,Y -45.308,Z -109.158,A -90.000,B 90.000,C 0.000} C_DIS
LIN {X -8.581,Y -45.308,Z -108.460,A -90.000,B 90.000,C 0.000} C_DIS
LIN {X -9.145,Y -45.308,Z -107.025,A -90.000,B 90.000,C 0.000} C_DIS
LIN {X -10.154,Y -45.308,Z -105.133,A -90.000,B 90.000,C 0.000} C_DIS
LIN {X -10.221,Y -45.308,Z -104.952,A -90.000,B 90.000,C 0.000} C_DIS
LIN {X -10.262,Y -45.308,Z -104.850,A -90.000,B 90.000,C 0.000} C_DIS
LIN {X -11.005,Y -45.308,Z -102.728,A -90.000,B 90.000,C 0.000} C_DIS
LIN {X -11.313,Y -45.308,Z -101.603,A -90.000,B 90.000,C 0.000} C_DIS
LIN {X -11.561,Y -45.308,Z -99.469,A -90.000,B 90.000,C 0.000} C_DIS
LIN {X -11.656,Y -45.308,Z -99.021,A -90.000,B 90.000,C 0.000} C_DIS
LIN {X -11.667,Y -45.308,Z -98.842,A -90.000,B 90.000,C 0.000} C_DIS
LIN {X -11.628,Y -45.308,Z -98.667,A -90.000,B 90.000,C 0.000} C_DIS
LIN {X -11.101,Y -45.308,Z -96.878,A -90.000,B 90.000,C 0.000} C_DIS
LIN {X -10.964,Y -45.308,Z -96.502,A -90.000,B 90.000,C 0.000} C_DIS
LIN {X -10.880,Y -45.308,Z -96.347,A -90.000,B 90.000,C 0.000} C_DIS
LIN {X -10.838,Y -45.308,Z -96.303,A -90.000,B 90.000,C 0.000} C_DIS
LIN {X -10.594,Y -45.308,Z -96.023,A -90.000,B 90.000,C 0.000} C_DIS
LIN {X -9.315,Y -45.308,Z -94.666,A -90.000,B 90.000,C 0.000} C_DIS
LIN {X -9.201,Y -45.308,Z -94.509,A -90.000,B 90.000,C 0.000} C_DIS
LIN {X -9.075,Y -45.308,Z -94.381,A -90.000,B 90.000,C 0.000} C_DIS
LIN {X -8.688,Y -45.308,Z -94.146,A -90.000,B 90.000,C 0.000} C_DIS
LIN {X -7.033,Y -45.308,Z -93.287,A -90.000,B 90.000,C 0.000} C_DIS
LIN {X -5.844,Y -45.308,Z -92.658,A -90.000,B 90.000,C 0.000} C_DIS
LIN {X -5.628,Y -45.308,Z -92.559,A -90.000,B 90.000,C 0.000} C_DIS
LIN {X -4.592,Y -45.308,Z -92.277,A -90.000,B 90.000,C 0.000} C_DIS
LIN {X -4.361,Y -45.308,Z -92.225,A -90.000,B 90.000,C 0.000} C_DIS
LIN {X -3.026,Y -45.308,Z -91.963,A -90.000,B 90.000,C 0.000} C_DIS
LIN {X -1.725,Y -45.308,Z -91.766,A -90.000,B 90.000,C 0.000} C_DIS
LIN {X -0.386,Y -45.308,Z -91.622,A -90.000,B 90.000,C 0.000} C_DIS
LIN {X 0.212,Y -45.308,Z -91.599,A -90.000,B 90.000,C 0.000} C_DIS
LIN {X 0.409,Y -45.314,Z -91.590,A -90.000,B 90.000,C 0.000} C_DIS
LIN {X 0.606,Y -45.312,Z -91.578,A -90.000,B 90.000,C 0.000} C_DIS
LIN {X 1.197,Y -45.303,Z -91.534,A -90.000,B 90.000,C 0.000} C_DIS
LIN {X 1.492,Y -45.295,Z -91.505,A -90.000,B 90.000,C 0.000} C_DIS
LIN {X 2.375,Y -45.266,Z -91.452,A -90.000,B 90.000,C 0.000} C_DIS
LIN {X 2.767,Y -45.249,Z -91.422,A -90.000,B 90.000,C 0.000} C_DIS
LIN {X 3.158,Y -45.230,Z -91.385,A -90.000,B 90.000,C 0.000} C_DIS
LIN {X 3.549,Y -45.208,Z -91.342,A -90.000,B 90.000,C 0.000} C_DIS
LIN {X 4.136,Y -45.174,Z -91.268,A -90.000,B 90.000,C 0.000} C_DIS
LIN {X 5.307,Y -45.097,Z -91.104,A -90.000,B 90.000,C 0.000} C_DIS
LIN {X 6.282,Y -45.034,Z -90.963,A -90.000,B 90.000,C 0.000} C_DIS
LIN {X 6.574,Y -45.015,Z -90.925,A -90.000,B 90.000,C 0.000} C_DIS
LIN {X 7.642,Y -44.945,Z -90.809,A -90.000,B 90.000,C 0.000} C_DIS
LIN {X 8.420,Y -44.895,Z -90.730,A -90.000,B 90.000,C 0.000} C_DIS
LIN {X 8.809,Y -44.870,Z -90.695,A -90.000,B 90.000,C 0.000} C_DIS
LIN {X 9.198,Y -44.844,Z -90.664,A -90.000,B 90.000,C 0.000} C_DIS
LIN {X 9.782,Y -44.807,Z -90.627,A -90.000,B 90.000,C 0.000} C_DIS
LIN {X 10.172,Y -44.781,Z -90.610,A -90.000,B 90.000,C 0.000} C_DIS
LIN {X 10.318,Y -44.772,Z -90.606,A -90.000,B 90.000,C 0.000} C_DIS
LIN {X 10.755,Y -44.744,Z -90.611,A -90.000,B 90.000,C 0.000} C_DIS
LIN {X 11.340,Y -44.706,Z -90.625,A -90.000,B 90.000,C 0.000} C_DIS
LIN {X 11.731,Y -44.681,Z -90.642,A -90.000,B 90.000,C 0.000} C_DIS
LIN {X 11.926,Y -44.668,Z -90.654,A -90.000,B 90.000,C 0.000} C_DIS
LIN {X 12.317,Y -44.643,Z -90.685,A -90.000,B 90.000,C 0.000} C_DIS
LIN {X 12.709,Y -44.617,Z -90.726,A -90.000,B 90.000,C 0.000} C_DIS
LIN {X 13.808,Y -44.613,Z -90.856,A -90.000,B 90.000,C 0.000} C_DIS
LIN {X 14.417,Y -44.608,Z -90.924,A -90.000,B 90.000,C 0.000} C_DIS
LIN {X 14.753,Y -44.608,Z -90.969,A -90.000,B 90.000,C 0.000} C_DIS
LIN {X 16.714,Y -44.626,Z -91.224,A -90.000,B 90.000,C 0.000} C_DIS
LIN {X 17.563,Y -44.626,Z -91.310,A -90.000,B 90.000,C 0.000} C_DIS
LIN {X 19.567,Y -44.647,Z -91.507,A -90.000,B 90.000,C 0.000} C_DIS
LIN {X 20.396,Y -44.640,Z -91.568,A -90.000,B 90.000,C 0.000} C_DIS
LIN {X 22.556,Y -44.651,Z -91.783,A -90.000,B 90.000,C 0.000} C_DIS
LIN {X 23.310,Y -44.644,Z -91.834,A -90.000,B 90.000,C 0.000} C_DIS
LIN {X 23.875,Y -44.651,Z -91.870,A -90.000,B 90.000,C 0.000} C_DIS
LIN {X 24.091,Y -44.655,Z -91.895,A -90.000,B 90.000,C 0.000} C_DIS
LIN {X 25.843,Y -44.673,Z -92.125,A -90.000,B 90.000,C 0.000} C_DIS
LIN {X 26.766,Y -44.671,Z -92.215,A -90.000,B 90.000,C 0.000} C_DIS
LIN {X 27.512,Y -44.683,Z -92.284,A -90.000,B 90.000,C 0.000} C_DIS
LIN {X 27.679,Y -44.689,Z -92.309,A -90.000,B 90.000,C 0.000} C_DIS
LIN {X 27.785,Y -44.693,Z -92.330,A -90.000,B 90.000,C 0.000} C_DIS
LIN {X 29.693,Y -44.722,Z -92.719,A -90.000,B 90.000,C 0.000} C_DIS
LIN {X 31.014,Y -44.727,Z -92.943,A -90.000,B 90.000,C 0.000} C_DIS
LIN {X 31.264,Y -44.732,Z -92.985,A -90.000,B 90.000,C 0.000} C_DIS
LIN {X 31.447,Y -44.737,Z -93.022,A -90.000,B 90.000,C 0.000} C_DIS
LIN {X 31.497,Y -44.737,Z -93.033,A -90.000,B 90.000,C 0.000} C_DIS
LIN {X 31.662,Y -44.740,Z -93.074,A -90.000,B 90.000,C 0.000} C_DIS
LIN {X 32.329,Y -44.748,Z -93.262,A -90.000,B 90.000,C 0.000} C_DIS
LIN {X 33.075,Y -44.746,Z -93.476,A -90.000,B 90.000,C 0.000} C_DIS
LIN {X 33.191,Y -44.746,Z -93.512,A -90.000,B 90.000,C 0.000} C_DIS
LIN {X 33.993,Y -44.758,Z -93.794,A -90.000,B 90.000,C 0.000} C_DIS
LIN {X 34.833,Y -44.773,Z -94.088,A -90.000,B 90.000,C 0.000} C_DIS
LIN {X 35.241,Y -44.772,Z -94.233,A -90.000,B 90.000,C 0.000} C_DIS
LIN {X 35.383,Y -44.771,Z -94.290,A -90.000,B 90.000,C 0.000} C_DIS
LIN {X 36.047,Y -44.771,Z -94.583,A -90.000,B 90.000,C 0.000} C_DIS
LIN {X 36.193,Y -44.772,Z -94.654,A -90.000,B 90.000,C 0.000} C_DIS
LIN {X 37.100,Y -44.794,Z -95.143,A -90.000,B 90.000,C 0.000} C_DIS
LIN {X 37.280,Y -44.798,Z -95.246,A -90.000,B 90.000,C 0.000} C_DIS
LIN {X 38.321,Y -44.805,Z -95.844,A -90.000,B 90.000,C 0.000} C_DIS
LIN {X 38.436,Y -44.807,Z -95.914,A -90.000,B 90.000,C 0.000} C_DIS
LIN {X 38.678,Y -44.812,Z -96.069,A -90.000,B 90.000,C 0.000} C_DIS
LIN {X 39.083,Y -44.811,Z -96.332,A -90.000,B 90.000,C 0.000} C_DIS
LIN {X 39.228,Y -44.813,Z -96.433,A -90.000,B 90.000,C 0.000} C_DIS
LIN {X 39.419,Y -44.813,Z -96.572,A -90.000,B 90.000,C 0.000} C_DIS
LIN {X 40.612,Y -44.816,Z -97.570,A -90.000,B 90.000,C 0.000} C_DIS
LIN {X 40.721,Y -44.817,Z -97.668,A -90.000,B 90.000,C 0.000} C_DIS
LIN {X 41.107,Y -44.827,Z -98.042,A -90.000,B 90.000,C 0.000} C_DIS
LIN {X 41.837,Y -44.825,Z -98.756,A -90.000,B 90.000,C 0.000} C_DIS
LIN {X 41.936,Y -44.823,Z -98.853,A -90.000,B 90.000,C 0.000} C_DIS
LIN {X 42.320,Y -44.808,Z -99.233,A -90.000,B 90.000,C 0.000} C_DIS
LIN {X 42.399,Y -44.806,Z -99.316,A -90.000,B 90.000,C 0.000} C_DIS
LIN {X 42.558,Y -44.802,Z -99.492,A -90.000,B 90.000,C 0.000} C_DIS
LIN {X 42.636,Y -44.802,Z -99.583,A -90.000,B 90.000,C 0.000} C_DIS
LIN {X 42.719,Y -44.802,Z -99.686,A -90.000,B 90.000,C 0.000} C_DIS
LIN {X 42.801,Y -44.803,Z -99.795,A -90.000,B 90.000,C 0.000} C_DIS
LIN {X 42.834,Y -44.804,Z -99.843,A -90.000,B 90.000,C 0.000} C_DIS
LIN {X 42.888,Y -44.805,Z -99.930,A -90.000,B 90.000,C 0.000} C_DIS
LIN {X 43.032,Y -44.808,Z -100.177,A -90.000,B 90.000,C 0.000} C_DIS
LIN {X 43.652,Y -44.831,Z -101.295,A -90.000,B 90.000,C 0.000} C_DIS
LIN {X 44.071,Y -44.831,Z -102.059,A -90.000,B 90.000,C 0.000} C_DIS
LIN {X 44.377,Y -44.831,Z -102.696,A -90.000,B 90.000,C 0.000} C_DIS
LIN {X 44.524,Y -44.817,Z -103.013,A -90.000,B 90.000,C 0.000} C_DIS
LIN {X 44.619,Y -44.806,Z -103.217,A -90.000,B 90.000,C 0.000} C_DIS
LIN {X 44.995,Y -44.763,Z -104.033,A -90.000,B 90.000,C 0.000} C_DIS
LIN {X 45.086,Y -44.755,Z -104.264,A -90.000,B 90.000,C 0.000} C_DIS
LIN {X 45.158,Y -44.752,Z -104.490,A -90.000,B 90.000,C 0.000} C_DIS
LIN {X 45.189,Y -44.751,Z -104.594,A -90.000,B 90.000,C 0.000} C_DIS
LIN {X 45.245,Y -44.755,Z -104.846,A -90.000,B 90.000,C 0.000} C_DIS
LIN {X 45.317,Y -44.757,Z -105.119,A -90.000,B 90.000,C 0.000} C_DIS
LIN {X 45.348,Y -44.759,Z -105.255,A -90.000,B 90.000,C 0.000} C_DIS
LIN {X 45.375,Y -44.765,Z -105.441,A -90.000,B 90.000,C 0.000} C_DIS
LIN {X 45.403,Y -44.775,Z -105.681,A -90.000,B 90.000,C 0.000} C_DIS
LIN {X 45.421,Y -44.777,Z -105.899,A -90.000,B 90.000,C 0.000} C_DIS
LIN {X 45.661,Y -44.772,Z -108.820,A -90.000,B 90.000,C 0.000} C_DIS
LIN {X 45.666,Y -44.773,Z -108.901,A -90.000,B 90.000,C 0.000} C_DIS
LIN {X 45.661,Y -44.777,Z -109.139,A -90.000,B 90.000,C 0.000} C_DIS
LIN {X 45.625,Y -44.791,Z -109.622,A -90.000,B 90.000,C 0.000} C_DIS
LIN {X 45.563,Y -44.784,Z -110.341,A -90.000,B 90.000,C 0.000} C_DIS
LIN {X 45.419,Y -44.746,Z -111.938,A -90.000,B 90.000,C 0.000} C_DIS
LIN {X 45.318,Y -44.728,Z -112.886,A -90.000,B 90.000,C 0.000} C_DIS
LIN {X 45.275,Y -44.729,Z -113.141,A -90.000,B 90.000,C 0.000} C_DIS
LIN {X 45.188,Y -44.737,Z -113.516,A -90.000,B 90.000,C 0.000} C_DIS
LIN {X 44.763,Y -44.705,Z -115.245,A -90.000,B 90.000,C 0.000} C_DIS
LIN {X 44.716,Y -44.704,Z -115.416,A -90.000,B 90.000,C 0.000} C_DIS
LIN {X 44.341,Y -44.695,Z -116.718,A -90.000,B 90.000,C 0.000} C_DIS
LIN {X 44.301,Y -44.696,Z -116.841,A -90.000,B 90.000,C 0.000} C_DIS
LIN {X 44.231,Y -44.699,Z -117.035,A -90.000,B 90.000,C 0.000} C_DIS
LIN {X 44.183,Y -44.701,Z -117.151,A -90.000,B 90.000,C 0.000} C_DIS
LIN {X 44.120,Y -44.704,Z -117.292,A -90.000,B 90.000,C 0.000} C_DIS
LIN {X 43.655,Y -44.701,Z -118.302,A -90.000,B 90.000,C 0.000} C_DIS
LIN {X 42.671,Y -44.700,Z -120.387,A -90.000,B 90.000,C 0.000} C_DIS
LIN {X 42.598,Y -44.702,Z -120.528,A -90.000,B 90.000,C 0.000} C_DIS
LIN {X 42.535,Y -44.704,Z -120.638,A -90.000,B 90.000,C 0.000} C_DIS
LIN {X 42.414,Y -44.705,Z -120.844,A -90.000,B 90.000,C 0.000} C_DIS
LIN {X 42.179,Y -44.705,Z -121.209,A -90.000,B 90.000,C 0.000} C_DIS
LIN {X 40.898,Y -44.678,Z -123.179,A -90.000,B 90.000,C 0.000} C_DIS
LIN {X 40.845,Y -44.677,Z -123.256,A -90.000,B 90.000,C 0.000} C_DIS
LIN {X 40.346,Y -44.672,Z -123.964,A -90.000,B 90.000,C 0.000} C_DIS
LIN {X 40.288,Y -44.670,Z -124.041,A -90.000,B 90.000,C 0.000} C_DIS
LIN {X 40.167,Y -44.667,Z -124.192,A -90.000,B 90.000,C 0.000} C_DIS
LIN {X 38.705,Y -44.612,Z -126.002,A -90.000,B 90.000,C 0.000} C_DIS
LIN {X 38.481,Y -44.608,Z -126.263,A -90.000,B 90.000,C 0.000} C_DIS
LIN {X 37.708,Y -44.606,Z -127.119,A -90.000,B 90.000,C 0.000} C_DIS
LIN {X 36.598,Y -44.563,Z -128.326,A -90.000,B 90.000,C 0.000} C_DIS
LIN {X 36.116,Y -44.542,Z -128.846,A -90.000,B 90.000,C 0.000} C_DIS
LIN {X 36.022,Y -44.540,Z -128.942,A -90.000,B 90.000,C 0.000} C_DIS
LIN {X 35.154,Y -44.539,Z -129.773,A -90.000,B 90.000,C 0.000} C_DIS
LIN {X 34.945,Y -44.534,Z -129.970,A -90.000,B 90.000,C 0.000} C_DIS
LIN {X 33.509,Y -44.469,Z -131.418,A -90.000,B 90.000,C 0.000} C_DIS
LIN {X 32.940,Y -44.445,Z -131.986,A -90.000,B 90.000,C 0.000} C_DIS
LIN {X 32.847,Y -44.443,Z -132.074,A -90.000,B 90.000,C 0.000} C_DIS
LIN {X 31.586,Y -44.443,Z -133.199,A -90.000,B 90.000,C 0.000} C_DIS
LIN {X 29.666,Y -44.367,Z -135.103,A -90.000,B 90.000,C 0.000} C_DIS
LIN {X 29.555,Y -44.364,Z -135.202,A -90.000,B 90.000,C 0.000} C_DIS
LIN {X 29.255,Y -44.363,Z -135.454,A -90.000,B 90.000,C 0.000} C_DIS
LIN {X 27.451,Y -44.306,Z -137.095,A -90.000,B 90.000,C 0.000} C_DIS
LIN {X 27.055,Y -44.290,Z -137.454,A -90.000,B 90.000,C 0.000} C_DIS
LIN {X 26.920,Y -44.279,Z -137.570,A -90.000,B 90.000,C 0.000} C_DIS
LIN {X 26.801,Y -44.272,Z -137.667,A -90.000,B 90.000,C 0.000} C_DIS
LIN {X 26.519,Y -44.271,Z -137.870,A -90.000,B 90.000,C 0.000} C_DIS
LIN {X 24.246,Y -44.220,Z -139.581,A -90.000,B 90.000,C 0.000} C_DIS
LIN {X 24.044,Y -44.220,Z -139.725,A -90.000,B 90.000,C 0.000} C_DIS
LIN {X 23.958,Y -44.215,Z -139.783,A -90.000,B 90.000,C 0.000} C_DIS
LIN {X 23.807,Y -44.210,Z -139.875,A -90.000,B 90.000,C 0.000} C_DIS
LIN {X 23.480,Y -44.209,Z -140.060,A -90.000,B 90.000,C 0.000} C_DIS
LIN {X 21.635,Y -44.192,Z -141.127,A -90.000,B 90.000,C 0.000} C_DIS
LIN {X 21.210,Y -44.184,Z -141.370,A -90.000,B 90.000,C 0.000} C_DIS
LIN {X 20.980,Y -44.186,Z -141.493,A -90.000,B 90.000,C 0.000} C_DIS
LIN {X 20.759,Y -44.189,Z -141.609,A -90.000,B 90.000,C 0.000} C_DIS
LIN {X 20.686,Y -44.189,Z -141.640,A -90.000,B 90.000,C 0.000} C_DIS
LIN {X 17.982,Y -44.147,Z -142.709,A -90.000,B 90.000,C 0.000} C_DIS
LIN {X 17.478,Y -44.139,Z -142.906,A -90.000,B 90.000,C 0.000} C_DIS
LIN {X 17.147,Y -44.143,Z -143.025,A -90.000,B 90.000,C 0.000} C_DIS
LIN {X 17.037,Y -44.146,Z -143.061,A -90.000,B 90.000,C 0.000} C_DIS
LIN {X 16.831,Y -44.155,Z -143.123,A -90.000,B 90.000,C 0.000} C_DIS
LIN {X 14.548,Y -44.140,Z -143.731,A -90.000,B 90.000,C 0.000} C_DIS
LIN {X 13.596,Y -44.127,Z -143.979,A -90.000,B 90.000,C 0.000} C_DIS
LIN {X 13.223,Y -44.125,Z -144.073,A -90.000,B 90.000,C 0.000} C_DIS
LIN {X 13.133,Y -44.125,Z -144.094,A -90.000,B 90.000,C 0.000} C_DIS
LIN {X 12.718,Y -44.135,Z -144.181,A -90.000,B 90.000,C 0.000} C_DIS
LIN {X 12.354,Y -44.152,Z -144.245,A -90.000,B 90.000,C 0.000} C_DIS
LIN {X 11.746,Y -44.153,Z -144.333,A -90.000,B 90.000,C 0.000} C_DIS
LIN {X 8.558,Y -44.190,Z -144.753,A -90.000,B 90.000,C 0.000} C_DIS
LIN {X 8.440,Y -44.193,Z -144.766,A -90.000,B 90.000,C 0.000} C_DIS
LIN {X 8.090,Y -44.208,Z -144.794,A -90.000,B 90.000,C 0.000} C_DIS
LIN {X 7.969,Y -44.213,Z -144.801,A -90.000,B 90.000,C 0.000} C_DIS
LIN {X 7.681,Y -44.224,Z -144.814,A -90.000,B 90.000,C 0.000} C_DIS
LIN {X 7.591,Y -44.226,Z -144.817,A -90.000,B 90.000,C 0.000} C_DIS
LIN {X 6.822,Y -44.224,Z -144.832,A -90.000,B 90.000,C 0.000} C_DIS
LIN {X 3.889,Y -44.259,Z -144.824,A -90.000,B 90.000,C 0.000} C_DIS
LIN {X 3.751,Y -44.264,Z -144.820,A -90.000,B 90.000,C 0.000} C_DIS
LIN {X 3.401,Y -44.281,Z -144.799,A -90.000,B 90.000,C 0.000} C_DIS
LIN {X 3.225,Y -44.292,Z -144.780,A -90.000,B 90.000,C 0.000} C_DIS
LIN {X 3.158,Y -44.298,Z -144.771,A -90.000,B 90.000,C 0.000} C_DIS
LIN {X 2.819,Y -44.314,Z -144.715,A -90.000,B 90.000,C 0.000} C_DIS
LIN {X 1.631,Y -44.339,Z -144.500,A -90.000,B 90.000,C 0.000} C_DIS
LIN {X 0.059,Y -44.337,Z -144.271,A -90.000,B 90.000,C 0.000} C_DIS
LIN {X -0.695,Y -44.346,Z -144.166,A -90.000,B 90.000,C 0.000} C_DIS
LIN {X -0.855,Y -44.353,Z -144.136,A -90.000,B 90.000,C 0.000} C_DIS
LIN {X -1.081,Y -44.367,Z -144.085,A -90.000,B 90.000,C 0.000} C_DIS
LIN {X -1.165,Y -44.368,Z -144.064,A -90.000,B 90.000,C 0.000} C_DIS
LIN {X -1.325,Y -44.373,Z -144.017,A -90.000,B 90.000,C 0.000} C_DIS
LIN {X -1.414,Y -44.379,Z -143.986,A -90.000,B 90.000,C 0.000} C_DIS
LIN {X -2.974,Y -44.432,Z -143.379,A -90.000,B 90.000,C 0.000} C_DIS
LIN {X -4.756,Y -44.454,Z -142.755,A -90.000,B 90.000,C 0.000} C_DIS
LIN {X -4.921,Y -44.463,Z -142.690,A -90.000,B 90.000,C 0.000} C_DIS
LIN {X -5.167,Y -44.467,Z -142.585,A -90.000,B 90.000,C 0.000} C_DIS
LIN {X -5.252,Y -44.470,Z -142.545,A -90.000,B 90.000,C 0.000} C_DIS
LIN {X -5.386,Y -44.472,Z -142.468,A -90.000,B 90.000,C 0.000} C_DIS
LIN {X -5.714,Y -44.484,Z -142.264,A -90.000,B 90.000,C 0.000} C_DIS
LIN {X -7.130,Y -44.561,Z -141.331,A -90.000,B 90.000,C 0.000} C_DIS
LIN {X -7.723,Y -44.574,Z -140.930,A -90.000,B 90.000,C 0.000} C_DIS
LIN {X -8.542,Y -44.578,Z -140.415,A -90.000,B 90.000,C 0.000} C_DIS
LIN {X -8.598,Y -44.579,Z -140.378,A -90.000,B 90.000,C 0.000} C_DIS
LIN {X -8.653,Y -44.577,Z -140.336,A -90.000,B 90.000,C 0.000} C_DIS
LIN {X -8.754,Y -44.575,Z -140.252,A -90.000,B 90.000,C 0.000} C_DIS
LIN {X -8.991,Y -44.574,Z -140.041,A -90.000,B 90.000,C 0.000} C_DIS
LIN {X -9.054,Y -44.574,Z -139.980,A -90.000,B 90.000,C 0.000} C_DIS
LIN {X -9.106,Y -44.575,Z -139.926,A -90.000,B 90.000,C 0.000} C_DIS
LIN {X -10.144,Y -44.591,Z -138.797,A -90.000,B 90.000,C 0.000} C_DIS
LIN {X -10.231,Y -44.594,Z -138.696,A -90.000,B 90.000,C 0.000} C_DIS
LIN {X -10.408,Y -44.603,Z -138.477,A -90.000,B 90.000,C 0.000} C_DIS
LIN {X -10.498,Y -44.610,Z -138.358,A -90.000,B 90.000,C 0.000} C_DIS
LIN {X -10.904,Y -44.651,Z -137.778,A -90.000,B 90.000,C 0.000} C_DIS
LIN {X -11.067,Y -44.673,Z -137.524,A -90.000,B 90.000,C 0.000} C_DIS
LIN {X -11.220,Y -44.685,Z -137.277,A -90.000,B 90.000,C 0.000} C_DIS
LIN {X -11.572,Y -44.695,Z -136.700,A -90.000,B 90.000,C 0.000} C_DIS
LIN {X -11.639,Y -44.698,Z -136.580,A -90.000,B 90.000,C 0.000} C_DIS
LIN {X -11.726,Y -44.704,Z -136.385,A -90.000,B 90.000,C 0.000} C_DIS
LIN {X -11.846,Y -44.711,Z -136.081,A -90.000,B 90.000,C 0.000} C_DIS
LIN {X -12.038,Y -44.728,Z -135.543,A -90.000,B 90.000,C 0.000} C_DIS
LIN {X -12.259,Y -44.728,Z -134.907,A -90.000,B 90.000,C 0.000} C_DIS
LIN {X -12.345,Y -44.730,Z -134.643,A -90.000,B 90.000,C 0.000} C_DIS
LIN {X -12.383,Y -44.732,Z -134.515,A -90.000,B 90.000,C 0.000} C_DIS
LIN {X -12.416,Y -44.735,Z -134.373,A -90.000,B 90.000,C 0.000} C_DIS
LIN {X -12.442,Y -44.740,Z -134.228,A -90.000,B 90.000,C 0.000} C_DIS
LIN {X -12.620,Y -44.738,Z -133.154,A -90.000,B 90.000,C 0.000} C_DIS
LIN {X -12.678,Y -44.737,Z -132.798,A -90.000,B 90.000,C 0.000} C_DIS
LIN {X -12.718,Y -44.738,Z -132.492,A -90.000,B 90.000,C 0.000} C_DIS
LIN {X -12.727,Y -44.739,Z -132.412,A -90.000,B 90.000,C 0.000} C_DIS
LIN {X -12.735,Y -44.742,Z -132.289,A -90.000,B 90.000,C 0.000} C_DIS
LIN {X -12.740,Y -44.747,Z -132.103,A -90.000,B 90.000,C 0.000} C_DIS
LIN {X -12.742,Y -44.746,Z -131.988,A -90.000,B 90.000,C 0.000} C_DIS
LIN {X -12.736,Y -44.747,Z -131.795,A -90.000,B 90.000,C 0.000} C_DIS
LIN {X -12.685,Y -44.760,Z -131.127,A -90.000,B 90.000,C 0.000} C_DIS
LIN {X -12.664,Y -44.764,Z -130.910,A -90.000,B 90.000,C 0.000} C_DIS
LIN {X -12.562,Y -44.765,Z -129.934,A -90.000,B 90.000,C 0.000} C_DIS
LIN {X -12.508,Y -44.755,Z -129.441,A -90.000,B 90.000,C 0.000} C_DIS
LIN {X -12.491,Y -44.754,Z -129.332,A -90.000,B 90.000,C 0.000} C_DIS
LIN {X -12.393,Y -44.754,Z -128.791,A -90.000,B 90.000,C 0.000} C_DIS
LIN {X -12.301,Y -44.760,Z -128.271,A -90.000,B 90.000,C 0.000} C_DIS
LIN {X -12.250,Y -44.765,Z -128.051,A -90.000,B 90.000,C 0.000} C_DIS
LIN {X -12.171,Y -44.775,Z -127.784,A -90.000,B 90.000,C 0.000} C_DIS
LIN {X -12.067,Y -44.788,Z -127.455,A -90.000,B 90.000,C 0.000} C_DIS
LIN {X -11.892,Y -44.796,Z -126.914,A -90.000,B 90.000,C 0.000} C_DIS
LIN {X -11.566,Y -44.797,Z -125.718,A -90.000,B 90.000,C 0.000} C_DIS
LIN {X -11.343,Y -44.814,Z -124.888,A -90.000,B 90.000,C 0.000} C_DIS
LIN {X -11.275,Y -44.820,Z -124.661,A -90.000,B 90.000,C 0.000} C_DIS
LIN {X -11.250,Y -44.822,Z -124.581,A -90.000,B 90.000,C 0.000} C_DIS
LIN {X -11.205,Y -44.828,Z -124.458,A -90.000,B 90.000,C 0.000} C_DIS
LIN {X -11.160,Y -44.832,Z -124.325,A -90.000,B 90.000,C 0.000} C_DIS
LIN {X -11.133,Y -44.833,Z -124.246,A -90.000,B 90.000,C 0.000} C_DIS
LIN {X -10.840,Y -44.835,Z -123.399,A -90.000,B 90.000,C 0.000} C_DIS
LIN {X -10.511,Y -44.869,Z -122.427,A -90.000,B 90.000,C 0.000} C_DIS
LIN {X -10.421,Y -44.869,Z -121.932,A -90.000,B 90.000,C 0.000} C_DIS
LIN {X -10.367,Y -44.872,Z -121.706,A -90.000,B 90.000,C 0.000} C_DIS
LIN {X -10.301,Y -44.877,Z -121.485,A -90.000,B 90.000,C 0.000} C_DIS
LIN {X -10.250,Y -44.883,Z -121.336,A -90.000,B 90.000,C 0.000} C_DIS
LIN {X -10.202,Y -44.887,Z -121.210,A -90.000,B 90.000,C 0.000} C_DIS
LIN {X -10.138,Y -44.890,Z -121.046,A -90.000,B 90.000,C 0.000} C_DIS
LIN {X -9.697,Y -44.939,Z -119.902,A -90.000,B 90.000,C 0.000} C_DIS
LIN {X -9.540,Y -44.938,Z -118.861,A -90.000,B 90.000,C 0.000} C_DIS
LIN {X -9.511,Y -44.946,Z -118.667,A -90.000,B 90.000,C 0.000} C_DIS
LIN {X -9.446,Y -44.961,Z -118.348,A -90.000,B 90.000,C 0.000} C_DIS
LIN {X -9.401,Y -44.971,Z -118.188,A -90.000,B 90.000,C 0.000} C_DIS
LIN {X -9.349,Y -44.982,Z -118.043,A -90.000,B 90.000,C 0.000} C_DIS
LIN {X -9.231,Y -44.995,Z -117.749,A -90.000,B 90.000,C 0.000} C_DIS
LIN {X -9.112,Y -44.986,Z -116.407,A -90.000,B 90.000,C 0.000} C_DIS
LIN {X -9.054,Y -45.006,Z -115.929,A -90.000,B 90.000,C 0.000} C_DIS
LIN {X -9.058,Y -45.006,Z -115.891,A -90.000,B 90.000,C 0.000} C_DIS
LIN {X -9.069,Y -45.008,Z -115.712,A -90.000,B 90.000,C 0.000} C_DIS
LIN {X -9.071,Y -45.013,Z -115.489,A -90.000,B 90.000,C 0.000} C_DIS
LIN {X -9.035,Y -45.034,Z -114.764,A -90.000,B 90.000,C 0.000} C_DIS
LIN {X -8.995,Y -45.035,Z -114.025,A -90.000,B 90.000,C 0.000} C_DIS
LIN {X -8.980,Y -45.048,Z -113.716,A -90.000,B 90.000,C 0.000} C_DIS
LIN {X -9.285,Y -45.047,Z -112.636,A -90.000,B 90.000,C 0.000} C_DIS
LIN {X -9.337,Y -45.046,Z -112.392,A -90.000,B 90.000,C 0.000} C_DIS
LIN {X -9.353,Y -45.048,Z -112.253,A -90.000,B 90.000,C 0.000} C_DIS
LIN {X -9.388,Y -45.056,Z -111.822,A -90.000,B 90.000,C 0.000} C_DIS
LIN {X -9.681,Y -45.050,Z -111.188,A -90.000,B 90.000,C 0.000} C_DIS
LIN {X -9.734,Y -45.049,Z -111.052,A -90.000,B 90.000,C 0.000} C_DIS
LIN {X -9.792,Y -45.048,Z -110.887,A -90.000,B 90.000,C 0.000} C_DIS
LIN {X -9.841,Y -45.047,Z -110.731,A -90.000,B 90.000,C 0.000} C_DIS
LIN {X -10.093,Y -45.047,Z -109.881,A -90.000,B 90.000,C 0.000} C_DIS
LIN {X -10.253,Y -45.039,Z -109.551,A -90.000,B 90.000,C 0.000} C_DIS
LIN {X -10.372,Y -45.039,Z -109.309,A -90.000,B 90.000,C 0.000} C_DIS
LIN {X -10.422,Y -45.040,Z -109.192,A -90.000,B 90.000,C 0.000} C_DIS
LIN {X -10.949,Y -45.056,Z -107.858,A -90.000,B 90.000,C 0.000} C_DIS
LIN {X -11.302,Y -45.050,Z -107.196,A -90.000,B 90.000,C 0.000} C_DIS
LIN {X -11.909,Y -45.026,Z -106.050,A -90.000,B 90.000,C 0.000} C_DIS
LIN {X -12.010,Y -45.024,Z -105.823,A -90.000,B 90.000,C 0.000} C_DIS
LIN {X -12.130,Y -45.023,Z -105.504,A -90.000,B 90.000,C 0.000} C_DIS
LIN {X -12.714,Y -45.031,Z -103.839,A -90.000,B 90.000,C 0.000} C_DIS
LIN {X -12.874,Y -45.031,Z -103.382,A -90.000,B 90.000,C 0.000} C_DIS
LIN {X -12.899,Y -45.031,Z -103.306,A -90.000,B 90.000,C 0.000} C_DIS
LIN {X -12.988,Y -45.034,Z -102.987,A -90.000,B 90.000,C 0.000} C_DIS
LIN {X -13.237,Y -45.034,Z -102.079,A -90.000,B 90.000,C 0.000} C_DIS
LIN {X -13.273,Y -45.036,Z -101.896,A -90.000,B 90.000,C 0.000} C_DIS
LIN {X -13.371,Y -45.053,Z -101.075,A -90.000,B 90.000,C 0.000} C_DIS
LIN {X -13.392,Y -45.054,Z -100.903,A -90.000,B 90.000,C 0.000} C_DIS
LIN {X -13.412,Y -45.052,Z -100.720,A -90.000,B 90.000,C 0.000} C_DIS
LIN {X -13.508,Y -45.031,Z -99.873,A -90.000,B 90.000,C 0.000} C_DIS
LIN {X -13.517,Y -45.029,Z -99.790,A -90.000,B 90.000,C 0.000} C_DIS
LIN {X -13.591,Y -45.015,Z -99.435,A -90.000,B 90.000,C 0.000} C_DIS
LIN {X -13.621,Y -45.009,Z -99.241,A -90.000,B 90.000,C 0.000} C_DIS
LIN {X -13.640,Y -45.004,Z -98.959,A -90.000,B 90.000,C 0.000} C_DIS
LIN {X -13.639,Y -45.003,Z -98.709,A -90.000,B 90.000,C 0.000} C_DIS
LIN {X -13.597,Y -45.008,Z -98.412,A -90.000,B 90.000,C 0.000} C_DIS
LIN {X -13.543,Y -45.015,Z -98.170,A -90.000,B 90.000,C 0.000} C_DIS
LIN {X -13.494,Y -45.017,Z -97.999,A -90.000,B 90.000,C 0.000} C_DIS
LIN {X -13.231,Y -44.988,Z -97.122,A -90.000,B 90.000,C 0.000} C_DIS
LIN {X -12.994,Y -44.979,Z -96.321,A -90.000,B 90.000,C 0.000} C_DIS
LIN {X -12.954,Y -44.978,Z -96.202,A -90.000,B 90.000,C 0.000} C_DIS
LIN {X -12.806,Y -44.978,Z -95.797,A -90.000,B 90.000,C 0.000} C_DIS
LIN {X -12.770,Y -44.977,Z -95.709,A -90.000,B 90.000,C 0.000} C_DIS
LIN {X -12.735,Y -44.976,Z -95.634,A -90.000,B 90.000,C 0.000} C_DIS
LIN {X -12.611,Y -44.963,Z -95.407,A -90.000,B 90.000,C 0.000} C_DIS
LIN {X -12.458,Y -44.951,Z -95.172,A -90.000,B 90.000,C 0.000} C_DIS
LIN {X -12.325,Y -44.947,Z -95.012,A -90.000,B 90.000,C 0.000} C_DIS
LIN {X -12.293,Y -44.947,Z -94.978,A -90.000,B 90.000,C 0.000} C_DIS
LIN {X -12.045,Y -44.941,Z -94.695,A -90.000,B 90.000,C 0.000} C_DIS
LIN {X -11.900,Y -44.943,Z -94.541,A -90.000,B 90.000,C 0.000} C_DIS
LIN {X -10.974,Y -44.951,Z -93.557,A -90.000,B 90.000,C 0.000} C_DIS
LIN {X -10.905,Y -44.951,Z -93.483,A -90.000,B 90.000,C 0.000} C_DIS
LIN {X -10.831,Y -44.948,Z -93.407,A -90.000,B 90.000,C 0.000} C_DIS
LIN {X -10.766,Y -44.941,Z -93.320,A -90.000,B 90.000,C 0.000} C_DIS
LIN {X -10.671,Y -44.931,Z -93.207,A -90.000,B 90.000,C 0.000} C_DIS
LIN {X -10.575,Y -44.923,Z -93.108,A -90.000,B 90.000,C 0.000} C_DIS
LIN {X -10.475,Y -44.916,Z -93.008,A -90.000,B 90.000,C 0.000} C_DIS
LIN {X -10.366,Y -44.909,Z -92.907,A -90.000,B 90.000,C 0.000} C_DIS
LIN {X -10.298,Y -44.906,Z -92.851,A -90.000,B 90.000,C 0.000} C_DIS
LIN {X -10.130,Y -44.903,Z -92.732,A -90.000,B 90.000,C 0.000} C_DIS
LIN {X -9.708,Y -44.902,Z -92.474,A -90.000,B 90.000,C 0.000} C_DIS
LIN {X -9.590,Y -44.902,Z -92.407,A -90.000,B 90.000,C 0.000} C_DIS
LIN {X -8.420,Y -44.918,Z -91.797,A -90.000,B 90.000,C 0.000} C_DIS
LIN {X -8.010,Y -44.916,Z -91.585,A -90.000,B 90.000,C 0.000} C_DIS
LIN {X -6.710,Y -44.840,Z -90.918,A -90.000,B 90.000,C 0.000} C_DIS
LIN {X -6.442,Y -44.828,Z -90.796,A -90.000,B 90.000,C 0.000} C_DIS
LIN {X -6.137,Y -44.821,Z -90.687,A -90.000,B 90.000,C 0.000} C_DIS
LIN {X -5.701,Y -44.821,Z -90.569,A -90.000,B 90.000,C 0.000} C_DIS
LIN {X -5.100,Y -44.811,Z -90.408,A -90.000,B 90.000,C 0.000} C_DIS
LIN {X -4.972,Y -44.810,Z -90.378,A -90.000,B 90.000,C 0.000} C_DIS
LIN {X -4.787,Y -44.808,Z -90.336,A -90.000,B 90.000,C 0.000} C_DIS
LIN {X -3.961,Y -44.808,Z -90.173,A -90.000,B 90.000,C 0.000} C_DIS
LIN {X -3.399,Y -44.796,Z -90.066,A -90.000,B 90.000,C 0.000} C_DIS
LIN {X -3.316,Y -44.794,Z -90.052,A -90.000,B 90.000,C 0.000} C_DIS
LIN {X -2.969,Y -44.791,Z -90.001,A -90.000,B 90.000,C 0.000} C_DIS
LIN {X -2.577,Y -44.782,Z -89.943,A -90.000,B 90.000,C 0.000} C_DIS
LIN {X -2.013,Y -44.762,Z -89.863,A -90.000,B 90.000,C 0.000} C_DIS
LIN {X -1.930,Y -44.760,Z -89.853,A -90.000,B 90.000,C 0.000} C_DIS
LIN {X -0.591,Y -44.728,Z -89.719,A -90.000,B 90.000,C 0.000} C_DIS
LIN {X -0.460,Y -44.726,Z -89.710,A -90.000,B 90.000,C 0.000} C_DIS
LIN {X 0.206,Y -44.723,Z -89.685,A -90.000,B 90.000,C 0.000} C_DIS
LIN {X 0.760,Y -44.712,Z -89.667,A -90.000,B 90.000,C 0.000} C_DIS
LIN {X 1.450,Y -44.701,Z -89.655,A -90.000,B 90.000,C 0.000} C_DIS
LIN {X 1.556,Y -44.700,Z -89.656,A -90.000,B 90.000,C 0.000} C_DIS
LIN {X 2.041,Y -44.700,Z -89.673,A -90.000,B 90.000,C 0.000} C_DIS
LIN {X 2.733,Y -44.706,Z -89.713,A -90.000,B 90.000,C 0.000} C_DIS
LIN {X 3.602,Y -44.704,Z -89.767,A -90.000,B 90.000,C 0.000} C_DIS
LIN {X 4.244,Y -44.701,Z -89.808,A -90.000,B 90.000,C 0.000} C_DIS
LIN {X 4.946,Y -44.689,Z -89.856,A -90.000,B 90.000,C 0.000} C_DIS
LIN {X 6.304,Y -44.672,Z -89.969,A -90.000,B 90.000,C 0.000} C_DIS
LIN {X 6.505,Y -44.668,Z -89.987,A -90.000,B 90.000,C 0.000} C_DIS
LIN {X 7.984,Y -44.656,Z -90.162,A -90.000,B 90.000,C 0.000} C_DIS
LIN {X 10.303,Y -44.630,Z -90.422,A -90.000,B 90.000,C 0.000} C_DIS
LIN {X 10.935,Y -44.630,Z -90.513,A -90.000,B 90.000,C 0.000} C_DIS
LIN {X 12.154,Y -44.620,Z -90.660,A -90.000,B 90.000,C 0.000} C_DIS
LIN {X 12.709,Y -44.617,Z -90.726,A -90.000,B 90.000,C 0.000} C_DIS
LIN {X 12.709,Y -60.000,Z -90.726,A -90.000,B 90.000,C 0.000} C_DIS
LIN {X -1.633,Y -60.000,Z -145.694,A -90.000,B 90.000,C 0.000} C_DIS
LIN {X -1.633,Y -43.308,Z -145.694,A -90.000,B 90.000,C 0.000} C_DIS
LIN {X -1.871,Y -43.325,Z -145.630,A -90.000,B 90.000,C 0.000} C_DIS
LIN {X -1.955,Y -43.330,Z -145.603,A -90.000,B 90.000,C 0.000} C_DIS
LIN {X -3.593,Y -43.422,Z -144.991,A -90.000,B 90.000,C 0.000} C_DIS
LIN {X -5.325,Y -43.478,Z -144.405,A -90.000,B 90.000,C 0.000} C_DIS
LIN {X -5.439,Y -43.482,Z -144.364,A -90.000,B 90.000,C 0.000} C_DIS
LIN {X -5.749,Y -43.499,Z -144.241,A -90.000,B 90.000,C 0.000} C_DIS
LIN {X -5.867,Y -43.501,Z -144.190,A -90.000,B 90.000,C 0.000} C_DIS
LIN {X -6.068,Y -43.508,Z -144.097,A -90.000,B 90.000,C 0.000} C_DIS
LIN {X -6.131,Y -43.509,Z -144.063,A -90.000,B 90.000,C 0.000} C_DIS
LIN {X -6.338,Y -43.516,Z -143.945,A -90.000,B 90.000,C 0.000} C_DIS
LIN {X -6.660,Y -43.533,Z -143.748,A -90.000,B 90.000,C 0.000} C_DIS
LIN {X -7.448,Y -43.589,Z -143.239,A -90.000,B 90.000,C 0.000} C_DIS
LIN {X -8.706,Y -43.671,Z -142.420,A -90.000,B 90.000,C 0.000} C_DIS
LIN {X -9.311,Y -43.698,Z -142.054,A -90.000,B 90.000,C 0.000} C_DIS
LIN {X -9.557,Y -43.698,Z -141.898,A -90.000,B 90.000,C 0.000} C_DIS
LIN {X -9.679,Y -43.695,Z -141.810,A -90.000,B 90.000,C 0.000} C_DIS
LIN {X -9.793,Y -43.693,Z -141.722,A -90.000,B 90.000,C 0.000} C_DIS
LIN {X -9.946,Y -43.694,Z -141.595,A -90.000,B 90.000,C 0.000} C_DIS
LIN {X -10.185,Y -43.700,Z -141.387,A -90.000,B 90.000,C 0.000} C_DIS
LIN {X -10.306,Y -43.705,Z -141.275,A -90.000,B 90.000,C 0.000} C_DIS
LIN {X -10.415,Y -43.713,Z -141.168,A -90.000,B 90.000,C 0.000} C_DIS
LIN {X -10.974,Y -43.763,Z -140.589,A -90.000,B 90.000,C 0.000} C_DIS
LIN {X -11.505,Y -43.812,Z -140.038,A -90.000,B 90.000,C 0.000} C_DIS
LIN {X -11.640,Y -43.828,Z -139.892,A -90.000,B 90.000,C 0.000} C_DIS
LIN {X -11.914,Y -43.869,Z -139.570,A -90.000,B 90.000,C 0.000} C_DIS
LIN {X -12.049,Y -43.894,Z -139.398,A -90.000,B 90.000,C 0.000} C_DIS
LIN {X -12.134,Y -43.913,Z -139.283,A -90.000,B 90.000,C 0.000} C_DIS
LIN {X -12.322,Y -43.946,Z -139.024,A -90.000,B 90.000,C 0.000} C_DIS
LIN {X -12.362,Y -43.951,Z -138.967,A -90.000,B 90.000,C 0.000} C_DIS
LIN {X -12.509,Y -43.962,Z -138.752,A -90.000,B 90.000,C 0.000} C_DIS
LIN {X -13.011,Y -43.995,Z -137.942,A -90.000,B 90.000,C 0.000} C_DIS
LIN {X -13.216,Y -44.002,Z -137.603,A -90.000,B 90.000,C 0.000} C_DIS
LIN {X -13.284,Y -44.005,Z -137.482,A -90.000,B 90.000,C 0.000} C_DIS
LIN {X -13.347,Y -44.011,Z -137.361,A -90.000,B 90.000,C 0.000} C_DIS
LIN {X -13.483,Y -44.030,Z -137.062,A -90.000,B 90.000,C 0.000} C_DIS
LIN {X -13.632,Y -44.058,Z -136.700,A -90.000,B 90.000,C 0.000} C_DIS
LIN {X -13.647,Y -44.062,Z -136.660,A -90.000,B 90.000,C 0.000} C_DIS
LIN {X -13.737,Y -44.075,Z -136.413,A -90.000,B 90.000,C 0.000} C_DIS
LIN {X -14.054,Y -44.103,Z -135.530,A -90.000,B 90.000,C 0.000} C_DIS
LIN {X -14.111,Y -44.109,Z -135.362,A -90.000,B 90.000,C 0.000} C_DIS
LIN {X -14.195,Y -44.118,Z -135.102,A -90.000,B 90.000,C 0.000} C_DIS
LIN {X -14.240,Y -44.125,Z -134.941,A -90.000,B 90.000,C 0.000} C_DIS
LIN {X -14.275,Y -44.132,Z -134.799,A -90.000,B 90.000,C 0.000} C_DIS
LIN {X -14.299,Y -44.139,Z -134.692,A -90.000,B 90.000,C 0.000} C_DIS
LIN {X -14.345,Y -44.152,Z -134.438,A -90.000,B 90.000,C 0.000} C_DIS
LIN {X -14.448,Y -44.165,Z -133.841,A -90.000,B 90.000,C 0.000} C_DIS
LIN {X -14.573,Y -44.162,Z -133.075,A -90.000,B 90.000,C 0.000} C_DIS
LIN {X -14.595,Y -44.162,Z -132.909,A -90.000,B 90.000,C 0.000} C_DIS
LIN {X -14.630,Y -44.164,Z -132.631,A -90.000,B 90.000,C 0.000} C_DIS
LIN {X -14.641,Y -44.166,Z -132.512,A -90.000,B 90.000,C 0.000} C_DIS
LIN {X -14.653,Y -44.173,Z -132.253,A -90.000,B 90.000,C 0.000} C_DIS
LIN {X -14.657,Y -44.172,Z -131.959,A -90.000,B 90.000,C 0.000} C_DIS
LIN {X -14.647,Y -44.174,Z -131.656,A -90.000,B 90.000,C 0.000} C_DIS
LIN {X -14.614,Y -44.183,Z -131.221,A -90.000,B 90.000,C 0.000} C_DIS
LIN {X -14.593,Y -44.192,Z -130.927,A -90.000,B 90.000,C 0.000} C_DIS
LIN {X -14.534,Y -44.217,Z -130.299,A -90.000,B 90.000,C 0.000} C_DIS
LIN {X -14.456,Y -44.224,Z -129.534,A -90.000,B 90.000,C 0.000} C_DIS
LIN {X -14.425,Y -44.223,Z -129.239,A -90.000,B 90.000,C 0.000} C_DIS
LIN {X -14.397,Y -44.223,Z -129.040,A -90.000,B 90.000,C 0.000} C_DIS
LIN {X -14.220,Y -44.233,Z -128.040,A -90.000,B 90.000,C 0.000} C_DIS
LIN {X -14.183,Y -44.234,Z -127.842,A -90.000,B 90.000,C 0.000} C_DIS
LIN {X -14.126,Y -44.238,Z -127.599,A -90.000,B 90.000,C 0.000} C_DIS
LIN {X -14.096,Y -44.241,Z -127.487,A -90.000,B 90.000,C 0.000} C_DIS
LIN {X -14.022,Y -44.249,Z -127.239,A -90.000,B 90.000,C 0.000} C_DIS
LIN {X -13.844,Y -44.271,Z -126.675,A -90.000,B 90.000,C 0.000} C_DIS
LIN {X -13.745,Y -44.283,Z -126.360,A -90.000,B 90.000,C 0.000} C_DIS
LIN {X -13.715,Y -44.286,Z -126.248,A -90.000,B 90.000,C 0.000} C_DIS
LIN {X -13.651,Y -44.286,Z -126.014,A -90.000,B 90.000,C 0.000} C_DIS
LIN {X -13.514,Y -44.296,Z -125.502,A -90.000,B 90.000,C 0.000} C_DIS
LIN {X -13.215,Y -44.331,Z -124.375,A -90.000,B 90.000,C 0.000} C_DIS
LIN {X -13.133,Y -44.342,Z -124.096,A -90.000,B 90.000,C 0.000} C_DIS
LIN {X -13.072,Y -44.350,Z -123.907,A -90.000,B 90.000,C 0.000} C_DIS
LIN {X -13.035,Y -44.358,Z -123.802,A -90.000,B 90.000,C 0.000} C_DIS
LIN {X -12.972,Y -44.371,Z -123.608,A -90.000,B 90.000,C 0.000} C_DIS
LIN {X -12.852,Y -44.394,Z -123.249,A -90.000,B 90.000,C 0.000} C_DIS
LIN {X -12.407,Y -44.445,Z -121.930,A -90.000,B 90.000,C 0.000} C_DIS
LIN {X -12.341,Y -44.447,Z -121.561,A -90.000,B 90.000,C 0.000} C_DIS
LIN {X -12.322,Y -44.451,Z -121.470,A -90.000,B 90.000,C 0.000} C_DIS
LIN {X -12.269,Y -44.463,Z -121.243,A -90.000,B 90.000,C 0.000} C_DIS
LIN {X -12.241,Y -44.469,Z -121.137,A -90.000,B 90.000,C 0.000} C_DIS
LIN {X -12.165,Y -44.485,Z -120.876,A -90.000,B 90.000,C 0.000} C_DIS
LIN {X -12.081,Y -44.503,Z -120.626,A -90.000,B 90.000,C 0.000} C_DIS
LIN {X -12.030,Y -44.514,Z -120.490,A -90.000,B 90.000,C 0.000} C_DIS
LIN {X -11.934,Y -44.530,Z -120.238,A -90.000,B 90.000,C 0.000} C_DIS
LIN {X -11.607,Y -44.567,Z -119.389,A -90.000,B 90.000,C 0.000} C_DIS
LIN {X -11.585,Y -44.567,Z -119.243,A -90.000,B 90.000,C 0.000} C_DIS
LIN {X -11.458,Y -44.600,Z -118.368,A -90.000,B 90.000,C 0.000} C_DIS
LIN {X -11.439,Y -44.604,Z -118.256,A -90.000,B 90.000,C 0.000} C_DIS
LIN {X -11.373,Y -44.620,Z -117.937,A -90.000,B 90.000,C 0.000} C_DIS
LIN {X -11.348,Y -44.626,Z -117.830,A -90.000,B 90.000,C 0.000} C_DIS
LIN {X -11.296,Y -44.637,Z -117.641,A -90.000,B 90.000,C 0.000} C_DIS
LIN {X -11.248,Y -44.648,Z -117.491,A -90.000,B 90.000,C 0.000} C_DIS
LIN {X -11.170,Y -44.664,Z -117.280,A -90.000,B 90.000,C 0.000} C_DIS
LIN {X -11.155,Y -44.669,Z -117.101,A -90.000,B 90.000,C 0.000} C_DIS
LIN {X -11.136,Y -44.668,Z -116.880,A -90.000,B 90.000,C 0.000} C_DIS
LIN {X -11.083,Y -44.691,Z -116.235,A -90.000,B 90.000,C 0.000} C_DIS
LIN {X -11.041,Y -44.708,Z -115.872,A -90.000,B 90.000,C 0.000} C_DIS
LIN {X -11.047,Y -44.712,Z -115.718,A -90.000,B 90.000,C 0.000} C_DIS
LIN {X -11.048,Y -44.720,Z -115.417,A -90.000,B 90.000,C 0.000} C_DIS
LIN {X -10.976,Y -44.774,Z -113.938,A -90.000,B 90.000,C 0.000} C_DIS
LIN {X -11.191,Y -44.767,Z -113.174,A -90.000,B 90.000,C 0.000} C_DIS
LIN {X -11.221,Y -44.767,Z -113.053,A -90.000,B 90.000,C 0.000} C_DIS
LIN {X -11.273,Y -44.767,Z -112.808,A -90.000,B 90.000,C 0.000} C_DIS
LIN {X -11.290,Y -44.767,Z -112.721,A -90.000,B 90.000,C 0.000} C_DIS
LIN {X -11.305,Y -44.768,Z -112.616,A -90.000,B 90.000,C 0.000} C_DIS
LIN {X -11.327,Y -44.771,Z -112.420,A -90.000,B 90.000,C 0.000} C_DIS
LIN {X -11.334,Y -44.772,Z -112.331,A -90.000,B 90.000,C 0.000} C_DIS
LIN {X -11.423,Y -44.766,Z -112.136,A -90.000,B 90.000,C 0.000} C_DIS
LIN {X -11.471,Y -44.765,Z -112.033,A -90.000,B 90.000,C 0.000} C_DIS
LIN {X -11.522,Y -44.765,Z -111.915,A -90.000,B 90.000,C 0.000} C_DIS
LIN {X -11.590,Y -44.765,Z -111.740,A -90.000,B 90.000,C 0.000} C_DIS
LIN {X -11.657,Y -44.767,Z -111.553,A -90.000,B 90.000,C 0.000} C_DIS
LIN {X -11.740,Y -44.770,Z -111.293,A -90.000,B 90.000,C 0.000} C_DIS
LIN {X -11.944,Y -44.781,Z -110.609,A -90.000,B 90.000,C 0.000} C_DIS
LIN {X -12.180,Y -44.775,Z -110.121,A -90.000,B 90.000,C 0.000} C_DIS
LIN {X -12.243,Y -44.772,Z -109.975,A -90.000,B 90.000,C 0.000} C_DIS
LIN {X -12.378,Y -44.775,Z -109.636,A -90.000,B 90.000,C 0.000} C_DIS
LIN {X -12.750,Y -44.772,Z -108.689,A -90.000,B 90.000,C 0.000} C_DIS
LIN {X -13.190,Y -44.752,Z -107.858,A -90.000,B 90.000,C 0.000} C_DIS
LIN {X -13.655,Y -44.739,Z -106.981,A -90.000,B 90.000,C 0.000} C_DIS
LIN {X -13.706,Y -44.738,Z -106.880,A -90.000,B 90.000,C 0.000} C_DIS
LIN {X -13.818,Y -44.738,Z -106.627,A -90.000,B 90.000,C 0.000} C_DIS
LIN {X -13.862,Y -44.738,Z -106.522,A -90.000,B 90.000,C 0.000} C_DIS
LIN {X -13.982,Y -44.738,Z -106.202,A -90.000,B 90.000,C 0.000} C_DIS
LIN {X -14.204,Y -44.740,Z -105.571,A -90.000,B 90.000,C 0.000} C_DIS
LIN {X -14.743,Y -44.749,Z -104.036,A -90.000,B 90.000,C 0.000} C_DIS
LIN {X -14.793,Y -44.749,Z -103.882,A -90.000,B 90.000,C 0.000} C_DIS
LIN {X -14.993,Y -44.749,Z -103.161,A -90.000,B 90.000,C 0.000} C_DIS
LIN {X -15.143,Y -44.742,Z -102.609,A -90.000,B 90.000,C 0.000} C_DIS
LIN {X -15.170,Y -44.741,Z -102.500,A -90.000,B 90.000,C 0.000} C_DIS
LIN {X -15.224,Y -44.740,Z -102.221,A -90.000,B 90.000,C 0.000} C_DIS
LIN {X -15.236,Y -44.741,Z -102.139,A -90.000,B 90.000,C 0.000} C_DIS
LIN {X -15.335,Y -44.748,Z -101.305,A -90.000,B 90.000,C 0.000} C_DIS
LIN {X -15.472,Y -44.742,Z -100.112,A -90.000,B 90.000,C 0.000} C_DIS
LIN {X -15.501,Y -44.739,Z -99.974,A -90.000,B 90.000,C 0.000} C_DIS
LIN {X -15.537,Y -44.730,Z -99.795,A -90.000,B 90.000,C 0.000} C_DIS
LIN {X -15.583,Y -44.717,Z -99.498,A -90.000,B 90.000,C 0.000} C_DIS
LIN {X -15.595,Y -44.713,Z -99.379,A -90.000,B 90.000,C 0.000} C_DIS
LIN {X -15.615,Y -44.703,Z -99.061,A -90.000,B 90.000,C 0.000} C_DIS
LIN {X -15.617,Y -44.700,Z -98.951,A -90.000,B 90.000,C 0.000} C_DIS
LIN {X -15.615,Y -44.695,Z -98.701,A -90.000,B 90.000,C 0.000} C_DIS
LIN {X -15.594,Y -44.692,Z -98.427,A -90.000,B 90.000,C 0.000} C_DIS
LIN {X -15.542,Y -44.691,Z -98.068,A -90.000,B 90.000,C 0.000} C_DIS
LIN {X -15.523,Y -44.694,Z -97.973,A -90.000,B 90.000,C 0.000} C_DIS
LIN {X -15.451,Y -44.703,Z -97.657,A -90.000,B 90.000,C 0.000} C_DIS
LIN {X -15.405,Y -44.710,Z -97.494,A -90.000,B 90.000,C 0.000} C_DIS
LIN {X -15.355,Y -44.712,Z -97.323,A -90.000,B 90.000,C 0.000} C_DIS
LIN {X -14.892,Y -44.661,Z -95.779,A -90.000,B 90.000,C 0.000} C_DIS
LIN {X -14.829,Y -44.655,Z -95.584,A -90.000,B 90.000,C 0.000} C_DIS
LIN {X -14.728,Y -44.648,Z -95.308,A -90.000,B 90.000,C 0.000} C_DIS
LIN {X -14.649,Y -44.649,Z -95.092,A -90.000,B 90.000,C 0.000} C_DIS
LIN {X -14.581,Y -44.645,Z -94.928,A -90.000,B 90.000,C 0.000} C_DIS
LIN {X -14.511,Y -44.636,Z -94.779,A -90.000,B 90.000,C 0.000} C_DIS
LIN {X -14.474,Y -44.631,Z -94.708,A -90.000,B 90.000,C 0.000} C_DIS
LIN {X -14.351,Y -44.617,Z -94.483,A -90.000,B 90.000,C 0.000} C_DIS
LIN {X -14.270,Y -44.609,Z -94.347,A -90.000,B 90.000,C 0.000} C_DIS
LIN {X -14.080,Y -44.595,Z -94.057,A -90.000,B 90.000,C 0.000} C_DIS
LIN {X -13.972,Y -44.590,Z -93.915,A -90.000,B 90.000,C 0.000} C_DIS
LIN {X -13.842,Y -44.586,Z -93.759,A -90.000,B 90.000,C 0.000} C_DIS
LIN {X -13.756,Y -44.585,Z -93.662,A -90.000,B 90.000,C 0.000} C_DIS
LIN {X -13.489,Y -44.579,Z -93.360,A -90.000,B 90.000,C 0.000} C_DIS
LIN {X -13.337,Y -44.577,Z -93.199,A -90.000,B 90.000,C 0.000} C_DIS
LIN {X -12.855,Y -44.578,Z -92.688,A -90.000,B 90.000,C 0.000} C_DIS
LIN {X -12.705,Y -44.571,Z -92.530,A -90.000,B 90.000,C 0.000} C_DIS
LIN {X -12.339,Y -44.541,Z -92.152,A -90.000,B 90.000,C 0.000} C_DIS
LIN {X -12.282,Y -44.534,Z -92.080,A -90.000,B 90.000,C 0.000} C_DIS
LIN {X -12.186,Y -44.524,Z -91.966,A -90.000,B 90.000,C 0.000} C_DIS
LIN {X -12.094,Y -44.515,Z -91.864,A -90.000,B 90.000,C 0.000} C_DIS
LIN {X -11.998,Y -44.508,Z -91.765,A -90.000,B 90.000,C 0.000} C_DIS
LIN {X -11.819,Y -44.495,Z -91.588,A -90.000,B 90.000,C 0.000} C_DIS
LIN {X -11.654,Y -44.485,Z -91.437,A -90.000,B 90.000,C 0.000} C_DIS
LIN {X -11.561,Y -44.481,Z -91.359,A -90.000,B 90.000,C 0.000} C_DIS
LIN {X -11.436,Y -44.477,Z -91.263,A -90.000,B 90.000,C 0.000} C_DIS
LIN {X -11.278,Y -44.474,Z -91.151,A -90.000,B 90.000,C 0.000} C_DIS
LIN {X -11.194,Y -44.472,Z -91.094,A -90.000,B 90.000,C 0.000} C_DIS
LIN {X -10.685,Y -44.471,Z -90.783,A -90.000,B 90.000,C 0.000} C_DIS
LIN {X -10.527,Y -44.472,Z -90.693,A -90.000,B 90.000,C 0.000} C_DIS
LIN {X -10.325,Y -44.469,Z -90.589,A -90.000,B 90.000,C 0.000} C_DIS
LIN {X -9.123,Y -44.437,Z -89.975,A -90.000,B 90.000,C 0.000} C_DIS
LIN {X -8.911,Y -44.426,Z -89.868,A -90.000,B 90.000,C 0.000} C_DIS
LIN {X -7.619,Y -44.358,Z -89.202,A -90.000,B 90.000,C 0.000} C_DIS
LIN {X -7.529,Y -44.354,Z -89.159,A -90.000,B 90.000,C 0.000} C_DIS
LIN {X -7.260,Y -44.344,Z -89.037,A -90.000,B 90.000,C 0.000} C_DIS
LIN {X -7.113,Y -44.340,Z -88.977,A -90.000,B 90.000,C 0.000} C_DIS
LIN {X -6.731,Y -44.326,Z -88.842,A -90.000,B 90.000,C 0.000} C_DIS
LIN {X -6.645,Y -44.323,Z -88.818,A -90.000,B 90.000,C 0.000} C_DIS
LIN {X -5.641,Y -44.280,Z -88.557,A -90.000,B 90.000,C 0.000} C_DIS
LIN {X -5.567,Y -44.277,Z -88.538,A -90.000,B 90.000,C 0.000} C_DIS
LIN {X -5.221,Y -44.266,Z -88.461,A -90.000,B 90.000,C 0.000} C_DIS
LIN {X -4.264,Y -44.244,Z -88.277,A -90.000,B 90.000,C 0.000} C_DIS
LIN {X -3.807,Y -44.231,Z -88.191,A -90.000,B 90.000,C 0.000} C_DIS
LIN {X -3.646,Y -44.225,Z -88.164,A -90.000,B 90.000,C 0.000} C_DIS
LIN {X -3.258,Y -44.211,Z -88.108,A -90.000,B 90.000,C 0.000} C_DIS
LIN {X -2.144,Y -44.173,Z -87.953,A -90.000,B 90.000,C 0.000} C_DIS
LIN {X -1.072,Y -44.149,Z -87.845,A -90.000,B 90.000,C 0.000} C_DIS
LIN {X -0.800,Y -44.136,Z -87.820,A -90.000,B 90.000,C 0.000} C_DIS
LIN {X -0.599,Y -44.126,Z -87.807,A -90.000,B 90.000,C 0.000} C_DIS
LIN {X 0.686,Y -44.080,Z -87.771,A -90.000,B 90.000,C 0.000} C_DIS
LIN {X 1.405,Y -44.059,Z -87.761,A -90.000,B 90.000,C 0.000} C_DIS
LIN {X 1.591,Y -44.055,Z -87.763,A -90.000,B 90.000,C 0.000} C_DIS
LIN {X 2.103,Y -44.048,Z -87.783,A -90.000,B 90.000,C 0.000} C_DIS
LIN {X 3.102,Y -44.028,Z -87.851,A -90.000,B 90.000,C 0.000} C_DIS
LIN {X 5.008,Y -43.992,Z -87.982,A -90.000,B 90.000,C 0.000} C_DIS
LIN {X 6.651,Y -43.959,Z -88.122,A -90.000,B 90.000,C 0.000} C_DIS
LIN {X 7.810,Y -43.949,Z -88.259,A -90.000,B 90.000,C 0.000} C_DIS
LIN {X 8.192,Y -43.944,Z -88.305,A -90.000,B 90.000,C 0.000} C_DIS
LIN {X 10.133,Y -43.910,Z -88.527,A -90.000,B 90.000,C 0.000} C_DIS
LIN {X 10.502,Y -43.902,Z -88.569,A -90.000,B 90.000,C 0.000} C_DIS
LIN {X 11.128,Y -43.896,Z -88.661,A -90.000,B 90.000,C 0.000} C_DIS
LIN {X 14.015,Y -43.857,Z -89.016,A -90.000,B 90.000,C 0.000} C_DIS
LIN {X 14.600,Y -43.850,Z -89.083,A -90.000,B 90.000,C 0.000} C_DIS
LIN {X 16.318,Y -43.851,Z -89.311,A -90.000,B 90.000,C 0.000} C_DIS
LIN {X 16.930,Y -43.857,Z -89.390,A -90.000,B 90.000,C 0.000} C_DIS
LIN {X 17.549,Y -43.856,Z -89.453,A -90.000,B 90.000,C 0.000} C_DIS
LIN {X 18.834,Y -43.858,Z -89.584,A -90.000,B 90.000,C 0.000} C_DIS
LIN {X 19.725,Y -43.872,Z -89.670,A -90.000,B 90.000,C 0.000} C_DIS
LIN {X 20.525,Y -43.876,Z -89.724,A -90.000,B 90.000,C 0.000} C_DIS
LIN {X 21.088,Y -43.883,Z -89.777,A -90.000,B 90.000,C 0.000} C_DIS
LIN {X 22.686,Y -43.918,Z -89.925,A -90.000,B 90.000,C 0.000} C_DIS
LIN {X 24.000,Y -43.929,Z -90.009,A -90.000,B 90.000,C 0.000} C_DIS
LIN {X 24.108,Y -43.931,Z -90.018,A -90.000,B 90.000,C 0.000} C_DIS
LIN {X 24.301,Y -43.937,Z -90.040,A -90.000,B 90.000,C 0.000} C_DIS
LIN {X 26.059,Y -43.986,Z -90.259,A -90.000,B 90.000,C 0.000} C_DIS
LIN {X 27.693,Y -44.010,Z -90.409,A -90.000,B 90.000,C 0.000} C_DIS
LIN {X 27.816,Y -44.017,Z -90.423,A -90.000,B 90.000,C 0.000} C_DIS
LIN {X 28.006,Y -44.029,Z -90.449,A -90.000,B 90.000,C 0.000} C_DIS
LIN {X 28.173,Y -44.037,Z -90.481,A -90.000,B 90.000,C 0.000} C_DIS
LIN {X 29.251,Y -44.077,Z -90.692,A -90.000,B 90.000,C 0.000} C_DIS
